# B&R Automation Studio project A2019059_Linka_Power_CP (part 11)

```iecst
(***************P4 - Funkčný test A************************************)

TYPE
	P4_FunkcnyTestA_typ : 	STRUCT
		IN : P4_FunkcnyTestA_IN_typ;
		OUT : P4_FunkcnyTestA_OUT_typ;
		PAR : P4_FunkcnyTestA_PAR_typ;
		STAV : P4_FunkcnyTestA_STAV_typ;
		Automat : BOOL;
		Manual : BOOL;
		Reset : BOOL;
		KoniecCyklu : BOOL;
		RR_TestovanieFunkcnehoTestu : BOOL;
		RR_ZapniOdpruzenieKontaktov : BOOL;
		RR_VysunKontaktyTestera : BOOL;
		RR_ZatvorTester : BOOL;
		RR_OtvorTester : BOOL;
	END_STRUCT;
	P4_FunkcnyTestA_IN_typ : 	STRUCT
		PritomnostPaletky_S10 : BOOL; (*RFID snímač na IO-linku*)
		PrecitaneCisloPaletky_S10 : USINT; (*RFID snímač na IO-linku*)
		HorneKontakty_VYSUNUTE_MS25 : BOOL;
		HorneKontakty_ZASUNUTE_MS23 : BOOL;
		SpodneKontakty_VYSUNUTE_MS33 : BOOL;
		SpodneKontakty_ZASUNUTE_MS31 : BOOL;
		Centrovanie_VYSUNUTE_MS29 : BOOL;
		Centrovanie_ZASUNUTE_MS27 : BOOL;
		TypSpodnychKontaktov_4F : BOOL;
		TypSpodnychKontaktov_5F_5H : BOOL;
	END_STRUCT;
	P4_FunkcnyTestA_OUT_typ : 	STRUCT
		ZasunStoper_YV163 : BOOL;
		HorneKontakty_VYSUN_YV178 : BOOL;
		HorneKontakty_ZASUN_YV177 : BOOL;
		OdpruzenieKontaktov_ZAPNI_YV179 : BOOL;
		OdpruzenieKontaktov_VYPNI_YV180 : BOOL;
		SpodneKontakty_VYSUN_YV182 : BOOL;
		SpodneKontakty_ZASUN_YV181 : BOOL;
		VysunCentrovanie_YV183 : BOOL;
		ZasunCentrovanie_YV184 : BOOL;
		KontaktyTestera_VYSUN_YV171 : BOOL;
		KOM_PLC_OdosliFotkyNaServer : BOOL;
		KOM_PLC_VymazFotky : BOOL;
	END_STRUCT;
	P4_FunkcnyTestA_PAR_typ : 	STRUCT
		SnimacPaletky_IOLinkInputs : ARRAY[1..10]OF USINT;
		IndexPaletky : USINT;
		IndexPaletky_STRING : STRING[2];
	END_STRUCT;
	P4_FunkcnyTestA_STAV_typ : 	STRUCT
		PoINIT : BOOL;
		KOM_PLC_OdoslanieFotiek_OK : BOOL;
		KOM_PLC_VymazanieFotiek_OK : BOOL;
		Vysledok_FV_Testu : STRING[2]; (*OK alebo NG*)
		PrebiehaVyvezeniePaletky : BOOL;
		Tester_ON : BOOL;
	END_STRUCT;
END_TYPE

(***************P4 - Funkčný test B************************************)

TYPE
	P4_FunkcnyTestB_typ : 	STRUCT
		IN : P4_FunkcnyTestB_IN_typ;
		OUT : P4_FunkcnyTestB_OUT_typ;
		PAR : P4_FunkcnyTestB_PAR_typ;
		STAV : P4_FunkcnyTestB_STAV_typ;
		Automat : BOOL;
		Manual : BOOL;
		Reset : BOOL;
		KoniecCyklu : BOOL;
		RR_TestovanieFunkcnehoTestu : BOOL;
		RR_ZapniOdpruzenieKontaktov : BOOL;
		RR_VysunKontaktyTestera : BOOL;
		RR_ZatvorTester : BOOL;
		RR_OtvorTester : BOOL;
	END_STRUCT;
	P4_FunkcnyTestB_IN_typ : 	STRUCT
		PritomnostPaletky_S11 : BOOL; (*RFID snímač na IO-linku*)
		PrecitaneCisloPaletky_S11 : USINT; (*RFID snímač na IO-linku*)
		HorneKontakty_VYSUNUTE_MS26 : BOOL;
		HorneKontakty_ZASUNUTE_MS24 : BOOL;
		SpodneKontakty_VYSUNUTE_MS34 : BOOL;
		SpodneKontakty_ZASUNUTE_MS32 : BOOL;
		Centrovanie_VYSUNUTE_MS30 : BOOL;
		Centrovanie_ZASUNUTE_MS28 : BOOL;
		TypSpodnychKontaktov_4F : BOOL;
		TypSpodnychKontaktov_5F_5H : BOOL;
	END_STRUCT;
	P4_FunkcnyTestB_OUT_typ : 	STRUCT
		ZasunStoper_YV164 : BOOL;
		HorneKontakty_VYSUN_YV186 : BOOL;
		HorneKontakty_ZASUN_YV185 : BOOL;
		OdpruzenieKontaktov_ZAPNI_YV187 : BOOL;
		OdpruzenieKontaktov_VYPNI_YV188 : BOOL;
		SpodneKontakty_VYSUN_YV190 : BOOL;
		SpodneKontakty_ZASUN_YV189 : BOOL;
		VysunCentrovanie_YV191 : BOOL;
		ZasunCentrovanie_YV192 : BOOL;
		KontaktyTestera_VYSUN_YV172 : BOOL;
		KOM_PLC_OdosliFotkyNaServer : BOOL;
		KOM_PLC_VymazFotky : BOOL;
		KOM_StanicaA_StartTestovania : BOOL;
	END_STRUCT;
	P4_FunkcnyTestB_PAR_typ : 	STRUCT
		SnimacPaletky_IOLinkInputs : ARRAY[1..10]OF USINT;
		IndexPaletky : USINT;
		IndexPaletky_STRING : STRING[2];
	END_STRUCT;
	P4_FunkcnyTestB_STAV_typ : 	STRUCT
		PoINIT : BOOL;
		KOM_PLC_OdoslanieFotiek_OK : BOOL;
		KOM_PLC_VymazanieFotiek_OK : BOOL;
		Vysledok_FV_Testu : STRING[2]; (*OK alebo NG*)
		PrebiehaVyvezeniePaletky : BOOL;
		Tester_ON : BOOL;
	END_STRUCT;
END_TYPE

(***************P4 - Etiketovacka*************************************)

TYPE
	P4_Etiketovacka_typ : 	STRUCT
		IN : P4_Etiketovacka_IN_typ;
		OUT : P4_Etiketovacka_OUT_typ;
		PAR : P4_Etiketovacka_PAR_typ;
		STAV : P4_Etiketovacka_STAV_typ;
		Automat : BOOL;
		Manual : BOOL;
		Reset : BOOL;
		KoniecCyklu : BOOL;
		ServoZdvihuEtiketovania_M28 : Axis_Servo;
		RR_TestovanieEtiketovania : BOOL;
		RR_VysunAplikator : BOOL;
		RR_ZapniPrisavanie : BOOL;
	END_STRUCT;
	P4_Etiketovacka_IN_typ : 	STRUCT
		PritomnostPaletky_S12 : BOOL; (*RFID snímač na IO-linku*)
		PrecitaneCisloPaletky_S12 : USINT; (*RFID snímač na IO-linku*)
		Centrovanie_VYSUNUTE_IS54 : BOOL;
		Centrovanie_ZASUNUTE_IS55 : BOOL;
		ZdvihEtiketovania_RefSnimac_IS59 : BOOL;
		Aplikator_VYSUNUTY_MS36 : BOOL;
		Aplikator_ZASUNUTY_MS35 : BOOL;
		SnimacVakuaPrisavaniaEtikety_S32 : BOOL;
		NapajanieTlaciarne_OK : BOOL;
		Tlaciaren_ERROR : BOOL;
		Tlaciaren_READY : BOOL;
		Tlaciaren_DochadzaPaska : BOOL;
		PritlakPaskyOdisteny_IS84 : BOOL;
	END_STRUCT;
	P4_Etiketovacka_OUT_typ : 	STRUCT
		ZasunStoper_YV165 : BOOL;
		VysunCentrovanie_YV166 : BOOL;
		ZasunCentrovanie_YV167 : BOOL;
		Aplikator_VYSUN_YV173 : BOOL;
		Prisavanie_ZAPNI_YV175 : BOOL;
		Prisavanie_VYPNI_YV176 : BOOL;
		OfukEtikety_ZAPNI_YV174 : BOOL;
		KOM_PLC_OdosliFotkyNaServer : BOOL;
		KOM_PLC_VymazFotky : BOOL;
		Tlaciaren_START_Tlace : BOOL;
		Tlaciaren_RESET_Poruchy : BOOL;
	END_STRUCT;
	P4_Etiketovacka_PAR_typ : 	STRUCT
		ServoZdvihu_ZadanaPozicia : LREAL;
		ServoZdvihu_JoggRychlost : REAL;
		SnimacPaletky_IOLinkInputs : ARRAY[1..10]OF USINT;
		IndexPaletky : USINT;
		IndexPaletky_STRING : STRING[2];
		IndexFotky : USINT;
	END_STRUCT;
	P4_Etiketovacka_STAV_typ : 	STRUCT
		PoINIT : BOOL;
		ServoZdvihu_PoziciaDosiahnuta : BOOL;
		ServoZvihu_LimitSnimace_BUSY : BOOL;
		ServoZdvihu_HomingOK : BOOL;
		ServoZdvihu_BUSY : BOOL;
		Zdvih_AktualnaPozicia : LREAL;
		Zdvih_AktualnyMoment : REAL;
		Zdvih_AktualnaRychlost : REAL;
		Zdvih_JoggLimitDosiahnuty : BOOL;
		KOM_PLC_OdoslanieFotiek_OK : BOOL;
		KOM_PLC_VymazanieFotiek_OK : BOOL;
		OdoslanieFotiek_OK : BOOL;
		OdoslanieFotiek_Error : BOOL;
		VymazanieFotiek_OK : BOOL;
		VymazanieFotiek_Error : BOOL;
		PrebiehaVyvezeniePaletky : BOOL;
		PowerCP_ZhodaQRkodu_OK : BOOL;
		Etiketa_ZhodaQRkodu_OK : BOOL;
		TestovaciaSekvencia_BUSY : BOOL;
	END_STRUCT;
END_TYPE

(******************SkrutkovacieSety***********************)

TYPE
	P1_SkrutkovaciSetM5_typ : 	STRUCT
		Automat : BOOL;
		Manual : BOOL;
		Reset : BOOL;
		UkoncenieCyklu : BOOL;
		SkrutkaM5_Pripravena : BOOL;
		SkrutkaM5_Odobrata : BOOL;
	END_STRUCT;
	P1_SkrutkovaciSetK30_typ : 	STRUCT
		Automat : BOOL;
		Manual : BOOL;
		Reset : BOOL;
		UkoncenieCyklu : BOOL;
		Cistenie : BOOL;
		CistenieUkoncene : BOOL;
		SkrutkaK30_Pripravena : BOOL;
		SkrutkaK30_Odobrata : BOOL;
	END_STRUCT;
	P1_SkrutkovaciSetM4_typ : 	STRUCT
		Automat : BOOL;
		Manual : BOOL;
		Reset : BOOL;
		UkoncenieCyklu : BOOL;
		Cistenie : BOOL;
		CistenieUkoncene : BOOL;
		SkrutkaM4_Pripravena : BOOL;
		SkrutkaM4_Odobrata : BOOL;
	END_STRUCT;
	P2_SkrutkovaciSetM6_typ : 	STRUCT
		Automat : BOOL;
		Manual : BOOL;
		Reset : BOOL;
		UkoncenieCyklu : BOOL;
		Cistenie : BOOL;
		CistenieUkoncene : BOOL;
		SkrutkaM6_Pripravena : BOOL;
		SkrutkaM6_Odobrata : BOOL;
	END_STRUCT;
	P2_SkrutkovaciSetM5_typ : 	STRUCT
		Automat : BOOL;
		Manual : BOOL;
		Reset : BOOL;
		UkoncenieCyklu : BOOL;
		Cistenie : BOOL;
		CistenieUkoncene : BOOL;
		SkrutkaM5_Pripravena : BOOL;
		SkrutkaM5_Odobrata : BOOL;
	END_STRUCT;
	P2_SkrutkovaciSetM4_typ : 	STRUCT
		Automat : BOOL;
		Manual : BOOL;
		Reset : BOOL;
		UkoncenieCyklu : BOOL;
		Cistenie : BOOL;
		CistenieUkoncene : BOOL;
		SkrutkaM4_Pripravena : BOOL;
		SkrutkaM4_Odobrata : BOOL;
	END_STRUCT;
	P2_SkrutkovaciSetMaticaM4_typ : 	STRUCT
		Automat : BOOL;
		Manual : BOOL;
		Reset : BOOL;
		UkoncenieCyklu : BOOL;
		MaticaM4_Pripravena : BOOL;
		MaticaM4_Odobrata : BOOL;
	END_STRUCT;
	P3_SkrutkovaciSetK40_typ : 	STRUCT
		Automat : BOOL;
		Manual : BOOL;
		Reset : BOOL;
		UkoncenieCyklu : BOOL;
		Cistenie : BOOL;
		CistenieUkoncene : BOOL;
		SkrutkaK40_Pripravena : BOOL;
		SkrutkaK40_Odobrata : BOOL;
	END_STRUCT;
	P3_SkrutkovaciSetM5_typ : 	STRUCT
		Automat : BOOL;
		Manual : BOOL;
		Reset : BOOL;
		UkoncenieCyklu : BOOL;
		Cistenie : BOOL;
		CistenieUkoncene : BOOL;
		SkrutkaM5_Pripravena : BOOL;
		SkrutkaM5_Odobrata : BOOL;
	END_STRUCT;
END_TYPE

(*******************Devlink*****************************)

TYPE
	StrukturaNovehoNazvuAdresara_typ : 	STRUCT
		LINKA : STRING[10]; (*Názov linky PowerCP*)
		PRACOVISKO : STRING[10]; (*ST1,ST2,ST3 .......*)
		ROK : STRING[10]; (*YYYY*)
		DATUM : STRING[10]; (*YYYY_MM_SS*)
	END_STRUCT;
	StrukturaNovehoNazvuSuboru_typ : 	STRUCT
		DATUM : STRING[10]; (*YYYY_MM_DD*)
		CAS : STRING[8]; (*HH_MM_SS*)
		SERIAL : STRING[30]; (*Kód modelu*)
		INDEX : STRING[2]; (*1,2,3 ......*)
		RESULT : STRING[5]; (*PASS alebo FAIL*)
		Pripona : STRING[5]; (*.jpg*)
	END_STRUCT;
END_TYPE

(**************Skrutkovacky***************************)

TYPE
	SkrutkovackaAtlasCopco_typ : 	STRUCT
		RESET_Poruchy : BOOL;
		RESET_Vysledkov : BOOL;
		START_Skrutkovania : BOOL;
		START_Utahovania : BOOL;
		Stav_VysledokPotvrdeny : BOOL;
		Stav_EmergencyStop : BOOL;
		Stav_READY_to_START : BOOL;
		Stav_MANUAL : BOOL;
		Stav_UtahovanieUkoncene : BOOL;
		Stav_VysledokUtahovania_OK : BOOL;
		Stav_VysledokUtahovania_NG : BOOL;
		Stav_SmerOtacania_VPRED : BOOL;
		Stav_BUSY : BOOL;
		Stav_ControlerSwitch_ON : BOOL;
		Stav_Station_READY : BOOL;
		Stav_NastrojPripojeny : BOOL;
		Stav_NastrojUtahuje : BOOL;
		Stav_CisloAktualnehoProgramu : USINT;
		CisloZadanehoProgramu : USINT;
		VyslednyReport : STRING[5];
	END_STRUCT;
END_TYPE

(**************Ateq Leakage Testery******************)

TYPE
	AteqTester_typ : 	STRUCT
		START_Testovania : BOOL;
		RESET_Vysledkov : BOOL;
		ZMEN_Program : BOOL;
		CitajParametreTestera : BOOL;
		Stav_RESET_DONE : BOOL;
		Stav_START_DONE : BOOL;
		Stav_ZmenaProgramu_DONE : BOOL;
		Stav_ERROR : BOOL;
		Stav_READY : BOOL;
		Stav_BUSY : BOOL;
		Stav_CitanieParametrov_OK : BOOL;
		Stav_CitanieParametrov_ERROR : BOOL;
		CisloZadanehoProgramu : UINT;
		CisloAktualnehoProgramu : UINT;
		VysledokTestovania_OK : BOOL;
		VysledokTestovania_NG : BOOL;
		Profinet_PLC_INPUTS : ARRAY[1..100]OF USINT;
		Profinet_PLC_OUTPUTS : ARRAY[1..100]OF USINT;
		ReadParameter_1 : UINT;
		ReadParameter_2 : UINT;
		ReadParameter_3 : UINT;
		ReadParameter_4 : UINT;
		ReadParameter_5 : DINT;
		PocetCitanychParametrov : USINT;
		IdentifikaciaParametra_1 : USINT;
		IdentifikaciaParametra_2 : USINT;
		IdentifikaciaParametra_3 : USINT;
		IdentifikaciaParametra_4 : USINT;
		CasPnenia : REAL;
		CasStabilizacie : REAL;
		TlakPlnenia : REAL;
		Tolerancia : REAL;
		TlakUniku : REAL;
	END_STRUCT;
END_TYPE

(***************Etiketa********************************)

TYPE
	Etiketa_typ : 	STRUCT
		LocationCode : STRING[2]; (*KK*)
		PartIdentNumber : STRING[7]; (*SSSSSSS*)
		ChangeIndex : STRING[2]; (*II*)
		ProductionYear : STRING[2]; (*JJ*)
		Manufactured : STRING[1]; (*H*)
		DayOfProduction : STRING[3]; (*TTT*)
		AssemblyLine : STRING[1]; (*M*)
		DayProductionCounter : STRING[5]; (*PPPPP*)
		SuplierNumber : STRING[6]; (*LLLLLL*)
		PlantCode : STRING[2]; (*NN*)
		DataMetrix : STRING[31]; (*Vytváram ho z kodu modelu na pracovisku etiketovania*)
		TypModelu : STRING[8];
		CountryCode : STRING[2];
		DatumVyroby : STRING[8]; (*02.03.20*)
	END_STRUCT;
END_TYPE

(***************Komunikácia zo serverom********************)

TYPE
	KOM_Server_typ : 	STRUCT
		CMD : KOM_Server_CMD_typ;
		INPUTS : KOM_Server_INPUTS_typ;
		OUTPUTS : KOM_Server_OUTPUTS_typ;
		STATUS : KOM_Server_STATUS_typ;
	END_STRUCT;
	KOM_Server_CMD_typ : 	STRUCT
		VyziadajStavPaletky_TYP1 : BOOL;
		PriradQRkodFiltra_TYP3 : BOOL;
		VyziadajCisloEtikety_TYP0 : BOOL;
		OdosliStavPaletky_TYP2 : BOOL;
	END_STRUCT;
	KOM_Server_INPUTS_typ : 	STRUCT
		TYP_Prikazu : STRING[1]; (*Typ*)
		CisloStanice : STRING[5]; (*Stanica*)
		CisloPaletky : STRING[10]; (*RFID paletky*)
		QRkodPowerCP : STRING[30]; (*Master number*)
		QRkodFiltra : STRING[30]; (*DPS1*)
		ID_Operatora : STRING[80]; (*Operator*)
		Report : STRING[4000]; (*DATA  - Oddelené bodkočiarkou*)
		StavPaletky : STRING[4]; (*PASS alebo FAIL*)
		IndexPaletky : USINT;
	END_STRUCT;
	KOM_Server_OUTPUTS_typ : 	STRUCT
		TYP_Prikazu : STRING[1]; (*Typ*)
		CisloStanice : STRING[5]; (*Stanica*)
		CisloPaletky : STRING[10]; (*RFID paletky*)
		QRkodPowerCP : STRING[30]; (*Master number*)
		QRkodFiltra : STRING[30]; (*DPS1*)
		ID_Operatora : STRING[8]; (*Operator*)
		CisloEtikety : STRING[31];
		DruhCinnostiNaPaletke : STRING[20]; (*PRD;ST1 alebo SMP;CAL;ST1 alebo RST;HVT;ST1*)
		PovolenieCinnostiNaPaletke : STRING[2]; (*OK alebo NG*)
	END_STRUCT;
	KOM_Server_STATUS_typ : 	STRUCT
		KomunikaciaUkoncena : BOOL;
		KomunikaciaError : BOOL;
	END_STRUCT;
END_TYPE

(***************Vysledné reporty***************************)

TYPE
	Reports_typ : 	STRUCT
		Kamery : ReportKamery_typ;
		Skrutkovacky : ReportSkrutkovacky_typ;
		Zvaranie : ReportZvarania_typ;
		LeakageTest : ReportLeakageTest_typ;
	END_STRUCT;
	ReportKamery_typ : 	STRUCT
		P1_CAM2_KontrolaPaletky : STRING[5]; (*Výtah*)
		P1_CAM4_KontrolaPinovDPS : STRING[5]; (*Výtah*)
		P1_CAM6_KontrolaPaletky : STRING[5]; (*Srobovanie*)
		P2_CAM1_KontrolaTesnenia : STRING[5];
		P2_CAM17_KontrolaPaletky : STRING[5]; (*Zakladanie tesnenia*)
		P2_CAM9_KontrolaPaletky : STRING[5]; (*Srobovanie matice*)
		P2_CAM10_KontrolaPaletky : STRING[5]; (*Srobovanie*)
		P2_CAM11_KontrolaZvaru : STRING[5]; (*Zvaranie*)
		P2_CAM11_KontrolaPowerCP : STRING[5]; (*Zvaranie*)
		P2_CAM12_KontrolaPaletky : STRING[5];
		P3_CAM13_KontrolaPaletky : STRING[5]; (*Srobovanie*)
		P4_CAM15_KontrolaPaletky : STRING[5]; (*Etiketovačka*)
		P4_CAM16_KontrolaPaletky : STRING[5]; (*Výtah*)
	END_STRUCT;
	ReportSkrutkovacky_typ : 	STRUCT
		Moment_ToleranciaMAX : ReportSrobov_MomentTolerMAX_typ;
		Moment_ToleranciaMIN : ReportSrobov_MomentTolerMIN_typ;
		Moment_NameranaHodnota : ReportSrobov_NameranyMoment_typ;
		Uhol_ToleranciaMAX : ReportSrobov_UholTolerMAX_typ;
		Uhol_ToleranciaMIN : ReportSrobov_UholTolerMIN_typ;
		Uhol_NameranaHodnota : ReportSrobov_NameranyUhol_typ;
		VyskaSkrutkovania : ReportSrobov_VyskaSkrutkov_typ;
		CasSkrutkovania : ReportSrobov_CasSkrutkov_typ;
		VyslednyReport : ReportSrobov_VyslednyReport_typ;
	END_STRUCT;
	ReportZvarania_typ : 	STRUCT
		Vyska : ReportZvarania_Vyska_typ;
		Moment : ReportZvarania_Moment_typ;
		Frekvencia : STRING[10];
		VyslednyReport : STRING[5];
	END_STRUCT;
	ReportZvarania_Vyska_typ : 	STRUCT
		LavyZvar : STRING[10];
		PravyZvar : STRING[10];
	END_STRUCT;
	ReportZvarania_Moment_typ : 	STRUCT
		LavyZvar : STRING[4];
		PravyZvar : STRING[4];
	END_STRUCT;
	ReportSrobov_MomentTolerMAX_typ : 	STRUCT
		P1_LavaSkrutkaK30 : STRING[10];
		P1_PravaSkrutkaK30 : STRING[10];
		P1_ZadnaSkrutkaM4 : STRING[10];
		P1_PrednaSkrutkaM4 : STRING[10];
		P1_SkrutkaDPS_M4 : STRING[10];
		P1_LavaSkrutkaM5 : STRING[10];
		P1_PravaSkrutkaM5 : STRING[10];
		P1_StrednaSkrutkaM5 : STRING[10];
		P2_MaticaM4 : STRING[10];
		P2_LavaSkrutkaM6 : STRING[10];
		P2_PravaSkrutkaM6 : STRING[10];
		P2_LavaSkrutkaM4 : STRING[10];
		P2_PravaSkrutkaM4 : STRING[10];
		P2_LavaSkrutkaM5 : STRING[10];
		P2_PravaSkrutkaM5 : STRING[10];
		P2_StrednaSkrutkaM4 : STRING[10];
		P3_SkrutkaK40 : STRING[10];
		P3_SkrutkaM5 : STRING[10];
	END_STRUCT;
	ReportSrobov_MomentTolerMIN_typ : 	STRUCT
		P1_LavaSkrutkaK30 : STRING[10];
		P1_PravaSkrutkaK30 : STRING[10];
		P1_ZadnaSkrutkaM4 : STRING[10];
		P1_PrednaSkrutkaM4 : STRING[10];
		P1_SkrutkaDPS_M4 : STRING[10];
		P1_LavaSkrutkaM5 : STRING[10];
		P1_PravaSkrutkaM5 : STRING[10];
		P1_StrednaSkrutkaM5 : STRING[10];
		P2_MaticaM4 : STRING[10];
		P2_LavaSkrutkaM6 : STRING[10];
		P2_PravaSkrutkaM6 : STRING[10];
		P2_LavaSkrutkaM4 : STRING[10];
		P2_PravaSkrutkaM4 : STRING[10];
		P2_LavaSkrutkaM5 : STRING[10];
		P2_PravaSkrutkaM5 : STRING[10];
		P2_StrednaSkrutkaM4 : STRING[10];
		P3_SkrutkaK40 : STRING[10];
		P3_SkrutkaM5 : STRING[10];
	END_STRUCT;
	ReportSrobov_NameranyMoment_typ : 	STRUCT
		P1_LavaSkrutkaK30 : STRING[10];
		P1_PravaSkrutkaK30 : STRING[10];
		P1_ZadnaSkrutkaM4 : STRING[10];
		P1_PrednaSkrutkaM4 : STRING[10];
		P1_SkrutkaDPS_M4 : STRING[10];
		P1_LavaSkrutkaM5 : STRING[10];
		P1_PravaSkrutkaM5 : STRING[10];
		P1_StrednaSkrutkaM5 : STRING[10];
		P2_MaticaM4 : STRING[10];
		P2_LavaSkrutkaM6 : STRING[10];
		P2_PravaSkrutkaM6 : STRING[10];
		P2_LavaSkrutkaM4 : STRING[10];
		P2_PravaSkrutkaM4 : STRING[10];
		P2_LavaSkrutkaM5 : STRING[10];
		P2_PravaSkrutkaM5 : STRING[10];
		P2_StrednaSkrutkaM4 : STRING[10];
		P3_SkrutkaK40 : STRING[10];
		P3_SkrutkaM5 : STRING[10];
	END_STRUCT;
	ReportSrobov_UholTolerMAX_typ : 	STRUCT
		P1_LavaSkrutkaK30 : STRING[10];
		P1_PravaSkrutkaK30 : STRING[10];
		P1_ZadnaSkrutkaM4 : STRING[10];
		P1_PrednaSkrutkaM4 : STRING[10];
		P1_SkrutkaDPS_M4 : STRING[10];
		P1_LavaSkrutkaM5 : STRING[10];
		P1_PravaSkrutkaM5 : STRING[10];
		P1_StrednaSkrutkaM5 : STRING[10];
		P2_MaticaM4 : STRING[10];
		P2_LavaSkrutkaM6 : STRING[10];
		P2_PravaSkrutkaM6 : STRING[10];
		P2_LavaSkrutkaM4 : STRING[10];
		P2_PravaSkrutkaM4 : STRING[10];
		P2_LavaSkrutkaM5 : STRING[10];
		P2_PravaSkrutkaM5 : STRING[10];
		P2_StrednaSkrutkaM4 : STRING[10];
		P3_SkrutkaK40 : STRING[10];
		P3_SkrutkaM5 : STRING[10];
	END_STRUCT;
	ReportSrobov_UholTolerMIN_typ : 	STRUCT
		P1_LavaSkrutkaK30 : STRING[10];
		P1_PravaSkrutkaK30 : STRING[10];
		P1_ZadnaSkrutkaM4 : STRING[10];
		P1_PrednaSkrutkaM4 : STRING[10];
		P1_SkrutkaDPS_M4 : STRING[10];
		P1_LavaSkrutkaM5 : STRING[10];
		P1_PravaSkrutkaM5 : STRING[10];
		P1_StrednaSkrutkaM5 : STRING[10];
		P2_MaticaM4 : STRING[10];
		P2_LavaSkrutkaM6 : STRING[10];
		P2_PravaSkrutkaM6 : STRING[10];
		P2_LavaSkrutkaM4 : STRING[10];
		P2_PravaSkrutkaM4 : STRING[10];
		P2_LavaSkrutkaM5 : STRING[10];
		P2_PravaSkrutkaM5 : STRING[10];
		P2_StrednaSkrutkaM4 : STRING[10];
		P3_SkrutkaK40 : STRING[10];
		P3_SkrutkaM5 : STRING[10];
	END_STRUCT;
	ReportSrobov_NameranyUhol_typ : 	STRUCT
		P1_LavaSkrutkaK30 : STRING[10];
		P1_PravaSkrutkaK30 : STRING[10];
		P1_ZadnaSkrutkaM4 : STRING[10];
		P1_PrednaSkrutkaM4 : STRING[10];
		P1_SkrutkaDPS_M4 : STRING[10];
		P1_LavaSkrutkaM5 : STRING[10];
		P1_PravaSkrutkaM5 : STRING[10];
		P1_StrednaSkrutkaM5 : STRING[10];
		P2_MaticaM4 : STRING[10];
		P2_LavaSkrutkaM6 : STRING[10];
		P2_PravaSkrutkaM6 : STRING[10];
		P2_LavaSkrutkaM4 : STRING[10];
		P2_PravaSkrutkaM4 : STRING[10];
		P2_LavaSkrutkaM5 : STRING[10];
		P2_PravaSkrutkaM5 : STRING[10];
		P2_StrednaSkrutkaM4 : STRING[10];
		P3_SkrutkaK40 : STRING[10];
		P3_SkrutkaM5 : STRING[10];
	END_STRUCT;
	ReportSrobov_VyskaSkrutkov_typ : 	STRUCT
		P1_LavaSkrutkaK30 : STRING[10];
		P1_PravaSkrutkaK30 : STRING[10];
		P1_ZadnaSkrutkaM4 : STRING[10];
		P1_PrednaSkrutkaM4 : STRING[10];
		P1_SkrutkaDPS_M4 : STRING[10];
		P1_LavaSkrutkaM5 : STRING[10];
		P1_PravaSkrutkaM5 : STRING[10];
		P1_StrednaSkrutkaM5 : STRING[10];
		P2_MaticaM4 : STRING[10];
		P2_LavaSkrutkaM6 : STRING[10];
		P2_PravaSkrutkaM6 : STRING[10];
		P2_LavaSkrutkaM4 : STRING[10];
		P2_PravaSkrutkaM4 : STRING[10];
		P2_LavaSkrutkaM5 : STRING[10];
		P2_PravaSkrutkaM5 : STRING[10];
		P2_StrednaSkrutkaM4 : STRING[10];
		P3_SkrutkaK40 : STRING[10];
		P3_SkrutkaM5 : STRING[10];
	END_STRUCT;
	ReportSrobov_CasSkrutkov_typ : 	STRUCT
		P1_LavaSkrutkaK30 : STRING[10];
		P1_PravaSkrutkaK30 : STRING[10];
		P1_ZadnaSkrutkaM4 : STRING[10];
		P1_PrednaSkrutkaM4 : STRING[10];
		P1_SkrutkaDPS_M4 : STRING[10];
		P1_LavaSkrutkaM5 : STRING[10];
		P1_PravaSkrutkaM5 : STRING[10];
		P1_StrednaSkrutkaM5 : STRING[10];
		P2_MaticaM4 : STRING[10];
		P2_LavaSkrutkaM6 : STRING[10];
		P2_PravaSkrutkaM6 : STRING[10];
		P2_LavaSkrutkaM4 : STRING[10];
		P2_PravaSkrutkaM4 : STRING[10];
		P2_LavaSkrutkaM5 : STRING[10];
		P2_PravaSkrutkaM5 : STRING[10];
		P2_StrednaSkrutkaM4 : STRING[10];
		P3_SkrutkaK40 : STRING[10];
		P3_SkrutkaM5 : STRING[10];
	END_STRUCT;
	ReportSrobov_VyslednyReport_typ : 	STRUCT
		P1_LavaSkrutkaK30 : STRING[5];
		P1_PravaSkrutkaK30 : STRING[5];
		P1_ZadnaSkrutkaM4 : STRING[5];
		P1_PrednaSkrutkaM4 : STRING[5];
		P1_SkrutkaDPS_M4 : STRING[5];
		P1_LavaSkrutkaM5 : STRING[5];
		P1_PravaSkrutkaM5 : STRING[5];
		P1_StrednaSkrutkaM5 : STRING[5];
		P2_MaticaM4 : STRING[5];
		P2_LavaSkrutkaM6 : STRING[5];
		P2_PravaSkrutkaM6 : STRING[5];
		P2_LavaSkrutkaM4 : STRING[5];
		P2_PravaSkrutkaM4 : STRING[5];
		P2_LavaSkrutkaM5 : STRING[5];
		P2_PravaSkrutkaM5 : STRING[5];
		P2_StrednaSkrutkaM4 : STRING[5];
		P3_SkrutkaK40 : STRING[5];
		P3_SkrutkaM5 : STRING[5];
	END_STRUCT;
	ReportLeakageTest_typ : 	STRUCT
		CasPlnenia : RepLeakTest_CasPlnenia_typ;
		CasStabilizacie : RepLeakTest_CasStabilizacie_typ;
		TlakPlnenia : RepLeakTest_TlakPlnenia_typ;
		TlakPritlaku : RepLeakTest_TlakPritlaku_typ;
		ToleranciaPritlaku_MIN : RepLeakTest_TolPritlakuMIN_typ;
		ToleranciaPritlaku_MAX : RepLeakTest_TolPritlakuMAX_typ;
		ToleranciaTlakUniku_MIN : RepLeakTest_TolTlakUnikuMIN_typ;
		ToleranciaTlakUniku_MAX : RepLeakTest_TolTlakUnikuMAX_typ;
		TlakUniku : RepLeakTest_TlakUniku_typ;
		Tolerancia : RepLeakTest_Tolerancia_typ;
		VyslednyReport : RepLeakTest_VyslednyReport_typ;
	END_STRUCT;
	RepLeakTest_CasPlnenia_typ : 	STRUCT
		StanicaA : STRING[10];
		StanicaB : STRING[10];
	END_STRUCT;
	RepLeakTest_CasStabilizacie_typ : 	STRUCT
		StanicaA : STRING[10];
		StanicaB : STRING[10];
	END_STRUCT;
	RepLeakTest_TlakPlnenia_typ : 	STRUCT
		StanicaA : STRING[10];
		StanicaB : STRING[10];
	END_STRUCT;
	RepLeakTest_TlakPritlaku_typ : 	STRUCT
		StanicaA : STRING[10];
		StanicaB : STRING[10];
	END_STRUCT;
	RepLeakTest_TolPritlakuMIN_typ : 	STRUCT
		StanicaA : STRING[10];
		StanicaB : STRING[10];
	END_STRUCT;
	RepLeakTest_TolPritlakuMAX_typ : 	STRUCT
		StanicaA : STRING[10];
		StanicaB : STRING[10];
	END_STRUCT;
	RepLeakTest_TlakUniku_typ : 	STRUCT
		StanicaA : STRING[10];
		StanicaB : STRING[10];
	END_STRUCT;
	RepLeakTest_TolTlakUnikuMIN_typ : 	STRUCT
		StanicaA : STRING[10];
		StanicaB : STRING[10];
	END_STRUCT;
	RepLeakTest_TolTlakUnikuMAX_typ : 	STRUCT
		StanicaA : STRING[10];
		StanicaB : STRING[10];
	END_STRUCT;
	RepLeakTest_Tolerancia_typ : 	STRUCT
		StanicaA : STRING[10];
		StanicaB : STRING[10];
	END_STRUCT;
	RepLeakTest_VyslednyReport_typ : 	STRUCT
		StanicaA : STRING[5];
		StanicaB : STRING[5];
	END_STRUCT;
END_TYPE

(***************Posielanie fotiek na server**********************)

TYPE
	FTP_Kamery_typ : 	STRUCT
		CMD : FTP_Kamery_CMD_typ;
		INPUTS : FTP_Kamery_INPUTS_typ;
		STATUS : FTP_Kamery_STATUS_typ;
	END_STRUCT;
	FTP_Kamery_CMD_typ : 	STRUCT
		OdosliFotku : BOOL;
		VymazFotku : BOOL;
	END_STRUCT;
	FTP_Kamery_INPUTS_typ : 	STRUCT
		QRkodPowerCP : STRING[30]; (*Master number*)
		Result : STRING[5]; (*PASS alebo FAIL*)
		IndexFotky : STRING[2];
	END_STRUCT;
	FTP_Kamery_STATUS_typ : 	STRUCT
		KomunikaciaUkoncena : BOOL;
		KomunikaciaError : BOOL;
		CisloPoruchy : USINT;
		AdresarPrazdny : BOOL;
	END_STRUCT;
END_TYPE

(***************Meranie taktime********************************)

TYPE
	Taktime_typ : 	STRUCT
		CMD : Taktime_CMD_typ;
		OUTPUTS : Taktime_OUTPUTS_typ;
	END_STRUCT;
	Taktime_CMD_typ : 	STRUCT
		START_Merania_1 : BOOL;
		ZAPIS_Hodnot_1 : BOOL;
		STOP_Merania_1 : BOOL;
		START_Merania_2 : BOOL;
		ZAPIS_Hodnot_2 : BOOL;
		STOP_Merania_2 : BOOL;
	END_STRUCT;
	Taktime_OUTPUTS_typ : 	STRUCT
		NameraneHodiny_1 : UINT;
		NameraneMinuty_1 : UINT;
		NameraneSekundy_1 : UINT;
		NameraneMilisekundy_1 : UINT;
		NameraneHodiny_2 : UINT;
		NameraneMinuty_2 : UINT;
		NameraneSekundy_2 : UINT;
		NameraneMilisekundy_2 : UINT;
	END_STRUCT;
END_TYPE
```

### KameryGlobal.typ
```iecst
(************Kamera 1*******************)

TYPE
	CAM1_typ : 	STRUCT
		CMD : CAM1_Commands_typ;
		PAR : CAM1_Parametre_typ;
		STAV : CAM1_Status_typ;
		RESULT : CAM1_Results_typ;
		Profinet_PLC_INPUTS : ARRAY[0..100]OF USINT;
		Profinet_PLC_OUTPUTS : ARRAY[0..3]OF USINT;
	END_STRUCT;
	CAM1_Commands_typ : 	STRUCT
		Triger : BOOL;
		OdosliFotku : BOOL;
		VymazFotku : BOOL;
	END_STRUCT;
	CAM1_Parametre_typ : 	STRUCT
		ResultFotky : STRING[5];
	END_STRUCT;
	CAM1_Status_typ : 	STRUCT
		BUSY : BOOL;
		SWITCH : BOOL;
		READY : BOOL;
		OLD_SWITCH : BOOL;
		Results_READY : BOOL;
		Command_READY : BOOL;
		Command_ERROR : BOOL;
		Command_AKCEPTOVANY : BOOL;
	END_STRUCT;
	CAM1_Results_typ : 	STRUCT
		PritomnTesnenia_OK : BOOL;
		ZalozenieTesnenia_OK : BOOL;
		PritomnPowerCP_5H5F : BOOL;
		PritomnPowerCP_4F : BOOL;
	END_STRUCT;
END_TYPE

(*********Kamera 2***********)

TYPE
	CAM2_typ : 	STRUCT
		CMD : CAM2_Commands_typ;
		PAR : CAM2_Parametre_typ;
		STAV : CAM2_Status_typ;
		RESULT : CAM2_Results_typ;
		Profinet_PLC_INPUTS : ARRAY[0..100]OF USINT;
		Profinet_PLC_OUTPUTS : ARRAY[0..3]OF USINT;
	END_STRUCT;
	CAM2_Commands_typ : 	STRUCT
		Triger : BOOL;
		OdosliFotku : BOOL;
		VymazFotku : BOOL;
	END_STRUCT;
	CAM2_Parametre_typ : 	STRUCT
		ResultFotky : STRING[5];
	END_STRUCT;
	CAM2_Status_typ : 	STRUCT
		READY : BOOL;
		BUSY : BOOL;
		SWITCH : BOOL;
		OLD_SWITCH : BOOL;
		Results_READY : BOOL;
		Command_READY : BOOL;
		Command_ERROR : BOOL;
		Command_AKCEPTOVANY : BOOL;
	END_STRUCT;
	CAM2_Results_typ : 	STRUCT
		Paletka : CAM2_Paletka_typ;
		PowerCP : CAM2_PowerCP_typ;
	END_STRUCT;
	CAM2_PowerCP_typ : 	STRUCT
		New_Member : USINT;
	END_STRUCT;
	CAM2_Paletka_typ : 	STRUCT
		Pritom_PowerCP_5F : BOOL;
		Pritom_PowerCP_4F : BOOL;
		Pritom_PowerCP_5H : BOOL;
		Pritom_Busbar_SpodnyLavy_5H : BOOL;
		Pritom_Busbar_SpodnyPravy_5H : BOOL;
		Pritom_KrytuBusbarov_5H : BOOL;
		Pritom_DPS_4F5F : BOOL;
		Pritom_Busbaru_Spodny_5F : BOOL;
		Pritom_Busbaru_Spodny_4F : BOOL;
		Pritom_Foamu_4F5F : BOOL;
		Pritomn_Skeletonu_4F5F : BOOL;
		Pritomn_Skeletonu_5H : BOOL;
		Nepritomn_TopCoveru_4F : BOOL;
		Nepritomn_TopCoveru_5F5H : BOOL;
		Pritomn_LavyMVcase : BOOL;
		Pritomn_PravyMVcase : BOOL;
		OsadeniePlastuDPS_OK : BOOL;
		KompletSpodneBusbary_OK : BOOL;
	END_STRUCT;
END_TYPE

(***********Kamera 3****************)

TYPE
	CAM3_typ : 	STRUCT
		CMD : CAM3_Commands_typ;
		PAR : CAM3_Parametre_typ;
		STAV : CAM3_Status_typ;
		RESULT : CAM3_Results_typ;
		Profinet_QRkod_Znaky : ARRAY[0..31]OF USINT;
		Profinet_PLC_INPUTS : ARRAY[0..100]OF USINT;
		Profinet_PLC_OUTPUTS : ARRAY[0..3]OF USINT;
	END_STRUCT;
	CAM3_Commands_typ : 	STRUCT
		Triger : BOOL;
		OdosliFotku : BOOL;
		VymazFotku : BOOL;
	END_STRUCT;
	CAM3_Parametre_typ : 	STRUCT
		ResultFotky : STRING[5];
	END_STRUCT;
	CAM3_Status_typ : 	STRUCT
		BUSY : BOOL;
		SWITCH : BOOL;
		READY : BOOL;
		OLD_SWITCH : BOOL;
		Results_READY : BOOL;
	END_STRUCT;
	CAM3_Results_typ : 	STRUCT
		Paletka : CAM3_Paletka_typ;
		PowerCP : CAM3_PowerCP_typ;
	END_STRUCT;
	CAM3_PowerCP_typ : 	STRUCT
		New_Member : USINT;
	END_STRUCT;
	CAM3_Paletka_typ : 	STRUCT
		CitanieQRkodu_DPS_OK : BOOL;
		PrecitanyQRkod_DPS : STRING[32];
	END_STRUCT;
END_TYPE

(***********Kamera 4******************)

TYPE
	CAM4_typ : 	STRUCT
		CMD : CAM4_Commands_typ;
		PAR : CAM4_Parametre_typ;
		STAV : CAM4_Status_typ;
		RESULT : CAM4_Results_typ;
		Profinet_PLC_INPUTS : ARRAY[0..100]OF USINT;
		Profinet_PLC_OUTPUTS : ARRAY[0..3]OF USINT;
	END_STRUCT;
	CAM4_Commands_typ : 	STRUCT
		Triger : BOOL;
		OdosliFotku : BOOL;
		VymazFotku : BOOL;
	END_STRUCT;
	CAM4_Parametre_typ : 	STRUCT
		ResultFotky : STRING[5];
	END_STRUCT;
	CAM4_Status_typ : 	STRUCT
		READY : BOOL;
		BUSY : BOOL;
		SWITCH : BOOL;
		OLD_SWITCH : BOOL;
		Results_READY : BOOL;
		Command_READY : BOOL;
		Command_ERROR : BOOL;
		Command_AKCEPTOVANY : BOOL;
	END_STRUCT;
	CAM4_Results_typ : 	STRUCT
		Paletka : CAM4_Paletka_typ;
		PowerCP : CAM4_PowerCP_typ;
	END_STRUCT;
	CAM4_PowerCP_typ : 	STRUCT
		New_Member : USINT;
	END_STRUCT;
	CAM4_Paletka_typ : 	STRUCT
		Pritomn_Pinu1_KrytDPS_4F5F : BOOL;
		Pritomn_Pinu2_KrytDPS_4F5F : BOOL;
		Pritomn_Pinu3_KrytDPS_4F5F : BOOL;
		Pritomn_Pinu4_KrytDPS_4F5F : BOOL;
		Pritomn_Pinu5_KrytDPS_4F5F : BOOL;
		Pritomn_Pinu6_KrytDPS_4F5F : BOOL;
		Pritom_DPS_4F5F : BOOL;
	END_STRUCT;
END_TYPE

(***********Kamera 5******************)

TYPE
	CAM5_typ : 	STRUCT
		CMD : CAM5_Commands_typ;
		PAR : CAM5_Parametre_typ;
		STAV : CAM5_Status_typ;
		RESULT : CAM5_Results_typ;
		Profinet_QRkod_Znaky : ARRAY[0..31]OF USINT;
		Profinet_PLC_INPUTS : ARRAY[0..100]OF USINT;
		Profinet_PLC_OUTPUTS : ARRAY[0..3]OF USINT;
	END_STRUCT;
	CAM5_Commands_typ : 	STRUCT
		Triger : BOOL;
		OdosliFotku : BOOL;
		VymazFotku : BOOL;
	END_STRUCT;
	CAM5_Parametre_typ : 	STRUCT
		ResultFotky : STRING[5];
	END_STRUCT;
	CAM5_Status_typ : 	STRUCT
		BUSY : BOOL;
		SWITCH : BOOL;
		READY : BOOL;
		OLD_SWITCH : BOOL;
		Results_READY : BOOL;
	END_STRUCT;
	CAM5_Results_typ : 	STRUCT
		Paletka : CAM5_Paletka_typ;
		PowerCP : CAM5_PowerCP_typ;
	END_STRUCT;
	CAM5_PowerCP_typ : 	STRUCT
		CitanieQRkodu_PowerCP_OK : BOOL;
		PrecitanyQRkod_PowerCP : STRING[32];
	END_STRUCT;
	CAM5_Paletka_typ : 	STRUCT
		New_Member : USINT;
	END_STRUCT;
END_TYPE

(***********Kamera 6********************)

TYPE
	CAM6_typ : 	STRUCT
		CMD : CAM6_Commands_typ;
		PAR : CAM6_Parametre_typ;
		STAV : CAM6_Status_typ;
		RESULT : CAM6_Results_typ;
		Profinet_PLC_INPUTS : ARRAY[0..100]OF USINT;
		Profinet_PLC_OUTPUTS : ARRAY[0..3]OF USINT;
	END_STRUCT;
	CAM6_Commands_typ : 	STRUCT
		Triger : BOOL;
		OdosliFotku : BOOL;
		VymazFotku : BOOL;
	END_STRUCT;
	CAM6_Parametre_typ : 	STRUCT
		ResultFotky : STRING[5];
	END_STRUCT;
	CAM6_Status_typ : 	STRUCT
		READY : BOOL;
		BUSY : BOOL;
		SWITCH : BOOL;
		OLD_SWITCH : BOOL;
		Results_READY : BOOL;
		Command_READY : BOOL;
		Command_ERROR : BOOL;
		Command_AKCEPTOVANY : BOOL;
	END_STRUCT;
	CAM6_Results_typ : 	STRUCT
		Paletka : CAM6_Paletka_typ;
		PowerCP : CAM6_PowerCP_typ;
	END_STRUCT;
	CAM6_PowerCP_typ : 	STRUCT
		Nepritom_LavyFoam_4F5F : BOOL;
		Nepritom_PravyFoam_4F5F : BOOL;
		Pritom_LavejSkrutkyK30 : BOOL;
		Pritom_PravejSkrutkyK30 : BOOL;
		Pritom_SkrutkyDPS_4F5F : BOOL;
		Nepritom_ZadnejSkrutkyM4_4F : BOOL;
		Nepritom_ZadnejSkrutkyM4_5F : BOOL;
		Nepritom_PrednejSkrutkyM4_4F : BOOL;
		Nepritom_PrednejSkrutkyM4_5F : BOOL;
		Pritom_LavejSkrutkyM5_5H : BOOL;
		Pritom_PravejSkrutkyM5_5H : BOOL;
		Pritom_StrednejSkrutkyM5_5H : BOOL;
	END_STRUCT;
	CAM6_Paletka_typ : 	STRUCT
		Pritom_SpodnychBusbarov_5H : BOOL;
		Pritom_KrytuBusbarov_5H : BOOL;
		Pritom_SpodnyBusbar_5F : BOOL;
		Pritom_SpodnyBusbar_4F : BOOL;
		Pritom_LavyFoam_4F5F : BOOL;
		Pritom_PravyFoam_4F5F : BOOL;
	END_STRUCT;
END_TYPE

(************Kamera 7*******************)

TYPE
	CAM7_typ : 	STRUCT
		CMD : CAM7_Commands_typ;
		PAR : CAM7_Parametre_typ;
		STAV : CAM7_Status_typ;
		RESULT : CAM7_Results_typ;
		Profinet_QRkod_Znaky : ARRAY[0..31]OF USINT;
		Profinet_PLC_INPUTS : ARRAY[0..100]OF USINT;
		Profinet_PLC_OUTPUTS : ARRAY[0..3]OF USINT;
	END_STRUCT;
	CAM7_Commands_typ : 	STRUCT
		Triger : BOOL;
		OdosliFotku : BOOL;
		VymazFotku : BOOL;
	END_STRUCT;
	CAM7_Parametre_typ : 	STRUCT
		ResultFotky : STRING[5];
	END_STRUCT;
	CAM7_Status_typ : 	STRUCT
		BUSY : BOOL;
		SWITCH : BOOL;
		READY : BOOL;
		OLD_SWITCH : BOOL;
		Results_READY : BOOL;
		Command_READY : BOOL;
		Command_ERROR : BOOL;
		Command_AKCEPTOVANY : BOOL;
	END_STRUCT;
	CAM7_Results_typ : 	STRUCT
		CitanieQRkodu_Filtra5H_OK : BOOL;
		PrecitanyQRkod_Filtra5H : STRING[32];
	END_STRUCT;
END_TYPE

(************Kamera 8********************)

TYPE
	CAM8_typ : 	STRUCT
		CMD : CAM8_Commands_typ;
		PAR : CAM8_Parametre_typ;
		STAV : CAM8_Status_typ;
		RESULT : CAM8_Results_typ;
		Profinet_QRkod_Znaky : ARRAY[0..31]OF USINT;
		Profinet_PLC_INPUTS : ARRAY[0..100]OF USINT;
		Profinet_PLC_OUTPUTS : ARRAY[0..3]OF USINT;
	END_STRUCT;
	CAM8_Commands_typ : 	STRUCT
		Triger : BOOL;
		OdosliFotku : BOOL;
		VymazFotku : BOOL;
	END_STRUCT;
	CAM8_Parametre_typ : 	STRUCT
		ResultFotky : STRING[5];
	END_STRUCT;
	CAM8_Status_typ : 	STRUCT
		BUSY : BOOL;
		SWITCH : BOOL;
		READY : BOOL;
		OLD_SWITCH : BOOL;
		Results_READY : BOOL;
	END_STRUCT;
	CAM8_Results_typ : 	STRUCT
		Paletka : CAM8_Paletka_typ;
		PowerCP : CAM8_PowerCP_typ;
	END_STRUCT;
	CAM8_PowerCP_typ : 	STRUCT
		CitanieQRkodu_PowerCP_OK : BOOL;
		PrecitanyQRkod_PowerCP : STRING[30];
	END_STRUCT;
	CAM8_Paletka_typ : 	STRUCT
		New_Member : USINT;
	END_STRUCT;
END_TYPE

(*************Kamera 9********************)

TYPE
	CAM9_typ : 	STRUCT
		CMD : CAM9_Commands_typ;
		PAR : CAM9_Parametre_typ;
		STAV : CAM9_Status_typ;
		RESULT : CAM9_Results_typ;
		Profinet_PLC_INPUTS : ARRAY[0..100]OF USINT;
		Profinet_PLC_OUTPUTS : ARRAY[0..3]OF USINT;
	END_STRUCT;
	CAM9_Commands_typ : 	STRUCT
		Triger : BOOL;
		OdosliFotku : BOOL;
		VymazFotku : BOOL;
	END_STRUCT;
	CAM9_Parametre_typ : 	STRUCT
		ResultFotky : STRING[5];
	END_STRUCT;
	CAM9_Status_typ : 	STRUCT
		BUSY : BOOL;
		SWITCH : BOOL;
		READY : BOOL;
		OLD_SWITCH : BOOL;
		Results_READY : BOOL;
	END_STRUCT;
	CAM9_Results_typ : 	STRUCT
		Paletka : CAM9_Paletka_typ;
		PowerCP : CAM9_PowerCP_typ;
	END_STRUCT;
	CAM9_PowerCP_typ : 	STRUCT
		NepritomMatice : BOOL;
		PritomnBusbaru_5H : BOOL;
	END_STRUCT;
	CAM9_Paletka_typ : 	STRUCT
		New_Member : USINT;
	END_STRUCT;
END_TYPE

(**************Kamera 10******************)

TYPE
	CAM10_typ : 	STRUCT
		CMD : CAM10_Commands_typ;
		PAR : CAM10_Parametre_typ;
		STAV : CAM10_Status_typ;
		RESULT : CAM10_Results_typ;
		Profinet_PLC_INPUTS : ARRAY[0..100]OF USINT;
		Profinet_PLC_OUTPUTS : ARRAY[0..3]OF USINT;
	END_STRUCT;
	CAM10_Commands_typ : 	STRUCT
		Triger : BOOL;
		OdosliFotku : BOOL;
		VymazFotku : BOOL;
	END_STRUCT;
	CAM10_Parametre_typ : 	STRUCT
		ResultFotky : STRING[5];
	END_STRUCT;
	CAM10_Status_typ : 	STRUCT
		BUSY : BOOL;
		SWITCH : BOOL;
		READY : BOOL;
		OLD_SWITCH : BOOL;
		Results_READY : BOOL;
		Command_READY : BOOL;
		Command_ERROR : BOOL;
		Command_AKCEPTOVANY : BOOL;
	END_STRUCT;
	CAM10_Results_typ : 	STRUCT
		Paletka : CAM10_Paletka_typ;
		PowerCP : CAM10_PowerCP_typ;
	END_STRUCT;
	CAM10_PowerCP_typ : 	STRUCT
		Pritomn_LavejSkrutkyM6_4F5F : BOOL;
		Pritomn_PravejSkrutkyM6_4F5F : BOOL;
		Pritomn_LavejM4_4F5F : BOOL;
		Pritomn_PravejM4_4F5F : BOOL;
		Pritomn_SkrutkyM4_Filtra_5H : BOOL;
		Pritomn_LavejSkrutkyM5_5H : BOOL;
		Pritomn_PravejSkrutkyM5_5H : BOOL;
	END_STRUCT;
	CAM10_Paletka_typ : 	STRUCT
		Pritomn_Busbarov_5F : BOOL;
		Pritomn_Busbarov_4F : BOOL;
		Pritomn_Busbarov_5H : BOOL;
		Pritomn_PowerCP_5H : BOOL;
		Pritomn_PowerCP_4F : BOOL;
		Pritomn_PowerCP_5F : BOOL;
	END_STRUCT;
END_TYPE

(**************Kamera 11*****************)

TYPE
	CAM11_typ : 	STRUCT
		CMD : CAM11_Commands_typ;
		PAR : CAM11_Parametre_typ;
		STAV : CAM11_Status_typ;
		RESULT : CAM11_Results_typ;
		Profinet_PLC_INPUTS : ARRAY[0..100]OF USINT;
		Profinet_PLC_OUTPUTS : ARRAY[0..3]OF USINT;
	END_STRUCT;
	CAM11_Commands_typ : 	STRUCT
		Triger : BOOL;
		OdosliFotku : BOOL;
		VymazFotku : BOOL;
	END_STRUCT;
	CAM11_Parametre_typ : 	STRUCT
		ResultFotky : STRING[5];
	END_STRUCT;
	CAM11_Status_typ : 	STRUCT
		BUSY : BOOL;
		SWITCH : BOOL;
		READY : BOOL;
		OLD_SWITCH : BOOL;
		Results_READY : BOOL;
		Command_READY : BOOL;
		Command_ERROR : BOOL;
		Command_AKCEPTOVANY : BOOL;
	END_STRUCT;
	CAM11_Results_typ : 	STRUCT
		Paletka : CAM11_Paletka_typ;
		PowerCP : CAM11_PowerCP_typ;
	END_STRUCT;
	CAM11_Paletka_typ : 	STRUCT
		New_Member : USINT;
	END_STRUCT;
	CAM11_PowerCP_typ : 	STRUCT
		Pritomn_PowerCP_4F : BOOL;
		Pritomn_PowerCP_5F : BOOL;
		Pritomn_PowerCP_5H : BOOL;
		Pritomn_LavyMVcase : BOOL;
		Pritomn_PravyMVcase : BOOL;
		LavyBusbar_Zvaranie_OK : BOOL;
		PravyBusbar_Zvaranie_OK : BOOL;
		Pritomn_TopCover_4F : BOOL;
		Pritomn_TopCover_5F : BOOL;
		Pritomn_TopCover_5H : BOOL;
	END_STRUCT;
END_TYPE

(***************Kamera 12*****************)

TYPE
	CAM12_typ : 	STRUCT
		CMD : CAM12_Commands_typ;
		PAR : CAM12_Parametre_typ;
		STAV : CAM12_Status_typ;
		RESULT : CAM12_Results_typ;
		Profinet_PLC_INPUTS : ARRAY[0..100]OF USINT;
		Profinet_PLC_OUTPUTS : ARRAY[0..3]OF USINT;
	END_STRUCT;
	CAM12_Commands_typ : 	STRUCT
		Triger : BOOL;
		OdosliFotku : BOOL;
		VymazFotku : BOOL;
	END_STRUCT;
	CAM12_Parametre_typ : 	STRUCT
		ResultFotky : STRING[5];
	END_STRUCT;
	CAM12_Status_typ : 	STRUCT
		BUSY : BOOL;
		SWITCH : BOOL;
		READY : BOOL;
		OLD_SWITCH : BOOL;
		Results_READY : BOOL;
		Command_READY : BOOL;
		Command_ERROR : BOOL;
		Command_AKCEPTOVANY : BOOL;
	END_STRUCT;
	CAM12_Results_typ : 	STRUCT
		Paletka : CAM12_Paletka_typ;
		PowerCP : CAM12_PowerCP_typ;
	END_STRUCT;
	CAM12_Paletka_typ : 	STRUCT
		Pritomn_TopCover_5H5F : BOOL;
		Pritomn_TopCover_4F : BOOL;
		Pritomn_LavyMVcase : BOOL;
		Pritomn_PravyMVcase : BOOL;
	END_STRUCT;
	CAM12_PowerCP_typ : 	STRUCT
		New_Member : USINT;
	END_STRUCT;
END_TYPE

(***************Kamera 13****************)

TYPE
	CAM13_typ : 	STRUCT
		CMD : CAM13_Commands_typ;
		PAR : CAM13_Parametre_typ;
		STAV : CAM13_Status_typ;
		RESULT : CAM13_Results_typ;
		Profinet_PLC_INPUTS : ARRAY[0..100]OF USINT;
		Profinet_PLC_OUTPUTS : ARRAY[0..3]OF USINT;
	END_STRUCT;
	CAM13_Commands_typ : 	STRUCT
		Triger : BOOL;
		OdosliFotku : BOOL;
		VymazFotku : BOOL;
	END_STRUCT;
	CAM13_Parametre_typ : 	STRUCT
		ResultFotky : STRING[5];
	END_STRUCT;
	CAM13_Status_typ : 	STRUCT
		BUSY : BOOL;
		SWITCH : BOOL;
		READY : BOOL;
		OLD_SWITCH : BOOL;
		Results_READY : BOOL;
		Command_READY : BOOL;
		Command_ERROR : BOOL;
		Command_AKCEPTOVANY : BOOL;
	END_STRUCT;
	CAM13_Results_typ : 	STRUCT
		Pritomn_SkrutkyK40_TopCover_4F5F : BOOL;
		Pritomn_SkrutkyM5_TopCover : BOOL;
	END_STRUCT;
END_TYPE

(***************Kamera 14*****************)

TYPE
	CAM14_typ : 	STRUCT
		CMD : CAM14_Commands_typ;
		PAR : CAM14_Parametre_typ;
		STAV : CAM14_Status_typ;
		RESULT : CAM14_Results_typ;
		Profinet_QRkod_Znaky : ARRAY[0..31]OF USINT;
		Profinet_PLC_INPUTS : ARRAY[0..100]OF USINT;
		Profinet_PLC_OUTPUTS : ARRAY[0..3]OF USINT;
	END_STRUCT;
	CAM14_Commands_typ : 	STRUCT
		Triger : BOOL;
		OdosliFotku : BOOL;
		VymazFotku : BOOL;
	END_STRUCT;
	CAM14_Parametre_typ : 	STRUCT
		ResultFotky : STRING[5];
	END_STRUCT;
	CAM14_Status_typ : 	STRUCT
		BUSY : BOOL;
		SWITCH : BOOL;
		READY : BOOL;
		OLD_SWITCH : BOOL;
		Results_READY : BOOL;
	END_STRUCT;
	CAM14_Results_typ : 	STRUCT
		Paletka : CAM14_Paletka_typ;
		PowerCP : CAM14_PowerCP_typ;
	END_STRUCT;
	CAM14_PowerCP_typ : 	STRUCT
		CitanieQRkodu_PowerCP_OK : BOOL;
		PrecitanyQRkod_PowerCP : STRING[32];
	END_STRUCT;
	CAM14_Paletka_typ : 	STRUCT
		New_Member : USINT;
	END_STRUCT;
END_TYPE

(****************Kamera 15***************)

TYPE
	CAM15_typ : 	STRUCT
		CMD : CAM15_Commands_typ;
		PAR : CAM15_Parametre_typ;
		STAV : CAM15_Status_typ;
		RESULT : CAM15_Results_typ;
		Profinet_QRkod_Znaky : ARRAY[0..31]OF USINT;
		Profinet_OCR_Znaky : ARRAY[0..31]OF USINT;
		Profinet_PLC_INPUTS : ARRAY[0..100]OF USINT;
		Profinet_PLC_OUTPUTS : ARRAY[0..3]OF USINT;
	END_STRUCT;
	CAM15_Commands_typ : 	STRUCT
		Triger : BOOL;
		OdosliFotku : BOOL;
		VymazFotku : BOOL;
	END_STRUCT;
	CAM15_Parametre_typ : 	STRUCT
		ResultFotky : STRING[5];
	END_STRUCT;
	CAM15_Status_typ : 	STRUCT
		BUSY : BOOL;
		SWITCH : BOOL;
		READY : BOOL;
		OLD_SWITCH : BOOL;
		Results_READY : BOOL;
		Command_READY : BOOL;
		Command_ERROR : BOOL;
		Command_AKCEPTOVANY : BOOL;
	END_STRUCT;
	CAM15_Results_typ : 	STRUCT
		Pritomn_Etikety : BOOL;
		Pritomn_LogoBMV : BOOL;
		Pritomn_Textu_PowerCP : BOOL;
		Pritomn_Textu_Panasonic : BOOL;
		Pritomn_Textu_SK : BOOL;
		CitanieQRkodu_Etikety_OK : BOOL;
		PrecitanyQRkod_Etikety : STRING[31];
		PrecitaneOCR_Etikety : STRING[32];
	END_STRUCT;
END_TYPE

(****************Kamera 16**************)

TYPE
	CAM16_typ : 	STRUCT
		CMD : CAM16_Commands_typ;
		PAR : CAM16_Parametre_typ;
		STAV : CAM16_Status_typ;
		RESULT : CAM16_Results_typ;
		Profinet_PLC_INPUTS : ARRAY[0..100]OF USINT;
		Profinet_PLC_OUTPUTS : ARRAY[0..3]OF USINT;
	END_STRUCT;
	CAM16_Commands_typ : 	STRUCT
		Triger : BOOL;
		OdosliFotku : BOOL;
		VymazFotku : BOOL;
	END_STRUCT;
	CAM16_Parametre_typ : 	STRUCT
		ResultFotky : STRING[5];
	END_STRUCT;
	CAM16_Status_typ : 	STRUCT
		BUSY : BOOL;
		SWITCH : BOOL;
		READY : BOOL;
		OLD_SWITCH : BOOL;
		Results_READY : BOOL;
		Command_READY : BOOL;
		Command_ERROR : BOOL;
		Command_AKCEPTOVANY : BOOL;
	END_STRUCT;
	CAM16_Results_typ : 	STRUCT
		New_Member : USINT;
		Paletka : CAM16_Paletka_typ;
		PowerCP : CAM16_PowerCP_typ;
	END_STRUCT;
	CAM16_Paletka_typ : 	STRUCT
		Pritomn_Busbarov_4F : BOOL;
		Pritomn_Busbarov_5F : BOOL;
		Pritomn_Busbarov_5H : BOOL;
		Pritomn_LavyMVcase : BOOL;
		Pritomn_PravyMVcase : BOOL;
		Pritomn_PowerCP : BOOL;
		PrazdnaPaletka : BOOL;
	END_STRUCT;
	CAM16_PowerCP_typ : 	STRUCT
		PritomnostSkrutky_K40 : BOOL;
		PritomnostSkrutky_M5 : BOOL;
	END_STRUCT;
END_TYPE

(*************Kamera 17*******************)

TYPE
	CAM17_typ : 	STRUCT
		CMD : CAM17_Commands_typ;
		PAR : CAM17_Parametre_typ;
		STAV : CAM17_Status_typ;
		RESULT : CAM17_Results_typ;
		Profinet_PLC_INPUTS : ARRAY[0..100]OF USINT;
		Profinet_PLC_OUTPUTS : ARRAY[0..3]OF USINT;
	END_STRUCT;
	CAM17_Commands_typ : 	STRUCT
		Triger : BOOL;
		OdosliFotku : BOOL;
		VymazFotku : BOOL;
	END_STRUCT;
	CAM17_Parametre_typ : 	STRUCT
		ResultFotky : STRING[5];
	END_STRUCT;
	CAM17_Status_typ : 	STRUCT
		BUSY : BOOL;
		SWITCH : BOOL;
		READY : BOOL;
		OLD_SWITCH : BOOL;
		Results_READY : BOOL;
		Command_READY : BOOL;
		Command_ERROR : BOOL;
		Command_AKCEPTOVANY : BOOL;
	END_STRUCT;
	CAM17_Results_typ : 	STRUCT
		Paletka : CAM17_Paletka_typ;
		PowerCP : CAM17_PowerCP_typ;
	END_STRUCT;
	CAM17_PowerCP_typ : 	STRUCT
		New_Member : USINT;
	END_STRUCT;
	CAM17_Paletka_typ : 	STRUCT
		Pritomn_TopCoveru_4F : BOOL;
		Pritomn_TopCoveru_5F : BOOL;
		Pritomn_TopCoveru_5H : BOOL;
		Pritomn_Busbary_5H : BOOL;
		Pritomn_Busbary_5F : BOOL;
		Pritomn_Busbary_4F : BOOL;
		Pritomn_LavyMVcase : BOOL;
		Pritomn_PravyMVcase : BOOL;
		Pritomn_PowerCP_4F : BOOL;
		Pritomn_PowerCP_5F : BOOL;
		Pritomn_PowerCP_5H : BOOL;
		PoziciaBusbarov4F5F_OK : BOOL;
		PoziciaBusbarov5H_OK : BOOL;
	END_STRUCT;
END_TYPE

(************Control Unit********************)

TYPE
	ControlUnit_typ : 	STRUCT
		Profinet_PLC_INPUTS : ARRAY[0..1]OF USINT;
		Stav_READY : BOOL;
	END_STRUCT;
END_TYPE
```

### Global.var - Global variables
```iecst
(**********Nastavenie času**************)
VAR
	DTSetTime_0 : DTSetTime;
	DTGetTime_0 : DTGetTime;
END_VAR
(**********Blikače*******************************)
VAR
	Blikac100ms : BOOL;
	Blikac200ms : BOOL;
	Blikac500ms : BOOL;
	Blikac1s : BOOL;
END_VAR
(**************Remanentné premenné*********)
VAR
	P1_RemPremenne : P1_RemPremenne_typ;
	P2_RemPremenne : P2_RemPremenne_typ;
	P34_RemPremenne : P34_RemPremenne_typ;
	MpRecipeXml_P1 : MpRecipeXml := (0);
	MpRecipeRegPar_P1 : MpRecipeRegPar := (0);
	MpRecipeUI_P1 : MpRecipeUI;
	P1_UlozPremenne : BOOL;
	P1_NacitajPremenne : BOOL;
	MpRecipeXml_P2 : MpRecipeXml := (0);
	MpRecipeRegPar_P2 : MpRecipeRegPar := (0);
	MpRecipeUI_P2 : MpRecipeUI;
	P2_UlozPremenne : BOOL;
	P2_NacitajPremenne : BOOL;
	MpRecipeXml_P34 : MpRecipeXml := (0);
	MpRecipeRegPar_P34 : MpRecipeRegPar := (0);
	MpRecipeUI_P34 : MpRecipeUI;
	P34_UlozPremenne : BOOL;
	P34_NacitajPremenne : BOOL;
END_VAR
VAR RETAIN
	P1_Skrutk_4F_LavaK30_Vysunutie : REAL;
	P1_Skrutk_4F_PravaK30_Vysunutie : REAL;
	P1_Skrutk_4F_ZadnaM4_Vysunutie : REAL;
	P1_Skrutk_4F_PrednaM4_Vysunutie : REAL;
	P1_Skrutk_4F_DPS_M4_Vysunutie : REAL;
	P1_Skrutk_5F_LavaK30_Vysunutie : REAL;
	P1_Skrutk_5F_PravaK30_Vysunutie : REAL;
	P1_Skrutk_5F_ZadnaM4_Vysunutie : REAL;
	P1_Skrutk_5F_PrednaM4_Vysunutie : REAL;
	P1_Skrutk_5F_DPS_M4_Vysunutie : REAL;
	P1_Skrutk_5H_LavaK30_Vysunutie : REAL;
	P1_Skrutk_5H_PravaK30_Vysunutie : REAL;
	P1_Skrutk_5H_LavaM5_Vysunutie : REAL;
	P1_Skrutk_5H_PravaM5_Vysunutie : REAL;
	P1_Skrutk_5H_StrednaM5_Vysunutie : REAL;
	P2_Skrutk_4F_LavaM6_Vysunutie : REAL;
	P2_Skrutk_4F_PravaM6_Vysunutie : REAL;
	P2_Skrutk_4F_LavaM4_Vysunutie : REAL;
	P2_Skrutk_4F_PravaM4_Vysunutie : REAL;
	P2_Skrutk_5F_LavaM6_Vysunutie : REAL;
	P2_Skrutk_5F_PravaM6_Vysunutie : REAL;
	P2_Skrutk_5F_LavaM4_Vysunutie : REAL;
	P2_Skrutk_5F_PravaM4_Vysunutie : REAL;
	P2_Skrutk_5H_LavaM5_Vysunutie : REAL;
	P2_Skrutk_5H_PravaM5_Vysunutie : REAL;
	P2_Skrutk_5H_StrednaM4_Vysunutie : REAL;
	P2_Maticovacka_5H_Vysunutie : REAL;
	P3_Skrutk_4F_StredK40_Vysunutie : REAL;
	P3_Skrutk_4F_StredM5_Vysunutie : REAL;
	P3_Skrutk_5F_StredK40_Vysunutie : REAL;
	P3_Skrutk_5F_StredM5_Vysunutie : REAL;
	P3_Skrutk_5H_StredM5_Vysunutie : REAL;
END_VAR
(*************Všeobecné premenné*************)
VAR
	FilterVizu_P1 : STRING[300];
	FilterVizu_P2 : STRING[300];
	FilterVizu_P34 : STRING[300];
	Vizu : Vizu_typ;
	P1_Vizu : P1_Vizu_typ;
	P2_Vizu : P2_Vizu_typ;
	P34_Vizu : P34_Vizu_typ;
END_VAR
VAR RETAIN
	Paletka : ARRAY[0..20] OF Paletka_typ;
END_VAR
VAR
	Etiketa : Etiketa_typ;
	Safety : Safety_typ;
	Linka : Linka_typ;
	Reports : Reports_typ;
	P1_Pracovisko : P1_Pracovisko_typ;
	SC_P1_Dopravniky : SequenceControlTyp;
	P1_Dopravniky : P1_Dopravniky_typ;
	SC_P1_SpodnyStoper : SequenceControlTyp;
	P1_SpodnyStoper : P1_SpodnyStoper_typ;
	SC_P1_Vytah : SequenceControlTyp;
	P1_Vytah : P1_Vytah_typ;
	SC_P1_StoperSrobovania : SequenceControlTyp;
	P1_StoperSrobovania : P1_StoperSrobovacky_typ;
	SC_P1_Srobovanie : SequenceControlTyp;
	P1_Srobovanie : P1_Srobovanie_typ;
	SC_P1_AkumulacnyStoper : SequenceControlTyp;
	P1_AkumulacnyStoper : P1_AkumulacnyStoper_typ;
	SC_P1_Robot : SequenceControlTyp;
	P1_Robot : P1_Robot_typ;
	P2_Pracovisko : P2_Pracovisko_typ;
	SC_P2_Dopravniky : SequenceControlTyp;
	P2_Dopravniky : P2_Dopravniky_typ;
	SC_P2_StoperZaklTesnenia : SequenceControlTyp;
	P2_StoperZaklTesnenia : P2_StoperZaklTesnenia_typ;
	SC_P2_ZakladacTesnenia : SequenceControlTyp;
	P2_ZakladacTesnenia : P2_ZakladacTesnenia_typ;
	SC_P2_StoperMaticovacky : SequenceControlTyp;
	P2_StoperMaticovacky : P2_StoperMaticovacky_typ;
	SC_P2_SkrutkovacMatic : SequenceControlTyp;
	P2_SkrutkovacMatic : P2_SkrutkovacMatic_typ;
	SC_P2_StoperSrobovania : SequenceControlTyp;
	P2_StoperSrobovania : P2_StoperSrobovania_typ;
	SC_P2_Srobovanie : SequenceControlTyp;
	P2_Srobovanie : P2_Srobovanie_typ;
	SC_P2_Robot : SequenceControlTyp;
	P2_Robot : P2_Robot_typ;
	SC_P2_StoperZvarania : SequenceControlTyp;
	P2_StoperZvarania : P2_StoperZvarania_typ;
	SC_P2_Zvaranie : SequenceControlTyp;
	P2_Zvaranie : P2_Zvaranie_typ;
	SC_P2_Cistenie : SequenceControlTyp;
	P2_Cistenie : P2_Cistenie_typ;
	P3_Pracovisko : P3_Pracovisko_typ;
	SC_P3_Dopravniky : SequenceControlTyp;
	P3_Dopravniky : P3_Dopravniky_typ;
	SC_P3_SpodnyStoper : SequenceControlTyp;
	P3_SpodnyStoper : P3_SpodnyStoper_typ;
	SC_P3_VstupnyStoper : SequenceControlTyp;
	P3_VstupnyStoper : P3_VstupnyStoper_typ;
	SC_P3_StoperSrobovania : SequenceControlTyp;
	P3_StoperSrobovania : P3_StoperSrobovania_typ;
	SC_P3_Srobovanie : SequenceControlTyp;
	P3_Srobovanie : P3_Srobovanie_typ;
	SC_P3_AkumulacnyStoper : SequenceControlTyp;
	P3_AkumulacnyStoper : P3_AkumulacnyStoper_typ;
	SC_P3_LeakageTestA : SequenceControlTyp;
	P3_LeakageTestA : P3_LeakageTestA_typ;
	AteqLeakageTester_A : AteqTester_typ;
	SC_P3_LeakageTestB : SequenceControlTyp;
	P3_LeakageTestB : P3_LeakageTestB_typ;
	AteqLeakageTester_B : AteqTester_typ;
	P4_Pracovisko : P4_Pracovisko_typ;
	SC_P4_Dopravniky : SequenceControlTyp;
	P4_Dopravniky : P4_Dopravniky_typ;
	SC_P4_Vytah : SequenceControlTyp;
	P4_Vytah : P4_Vytah_typ;
	SC_P4_FunkcnyTestA : SequenceControlTyp;
	P4_FunkcnyTestA : P4_FunkcnyTestA_typ;
	SC_P4_FunkcnyTestB : SequenceControlTyp;
	P4_FunkcnyTestB : P4_FunkcnyTestB_typ;
	SC_P4_Etiketovacka : SequenceControlTyp;
	P4_Etiketovacka : P4_Etiketovacka_typ;
END_VAR
(**********Príznaky**************************)
VAR
	P1_Srobovacky_VychodziaPozicia : BOOL;
	P2_Srobovacky_VychodziaPozicia : BOOL;
	P2_Srobov_ManipulaciaUkoncena : BOOL;
	P2_Zvaranie_ManipulaciaUkoncena : BOOL;
	P3_Srobovacky_VychodziaPozicia : BOOL;
	P3_LeakageTestA_VychodziaPozicia : BOOL;
	P3_LeakageTestB_VychodziaPozicia : BOOL;
	P4_FunkcnyTestA_VychodziaPozicia : BOOL;
	P4_FunkcnyTestB_VychodziaPozicia : BOOL;
	P4_Etiketovacka_VychodziaPozicia : BOOL;
	CasCakaniaNaDruhePracovisko : TIME;
	Cas_HVTester : TON;
	NameranyCas_InitTestera : TIME;
	NameranyCas_PoslanieQRkodu : TIME;
	NameranyCas_CelkovyCasTestovania : TIME;
	Cas_FunkcnyTestA : TON;
	Cas_FunkcnyTestB : TON;
	NameranyCasFunkcnehoTestuA : TIME;
	NameranyCasFunkcnehoTestuB : TIME;
	Cas_PresunuSkrutky : TON;
	NameranyCasPresunuSkrutky : TIME;
END_VAR
(*************Tracebility***********************)
VAR
	TRCB_P1_Vytah_ST1 : KOM_Server_typ;
	TRCB_P1_Srobovanie_ST2 : KOM_Server_typ;
	TRCB_P2_ZakladacTesnenia_ST3 : KOM_Server_typ;
	TRCB_P2_Maticovacka_ST4 : KOM_Server_typ;
	TRCB_P2_Srobovanie_ST5 : KOM_Server_typ;
	TRCB_P2_Zvaranie_ST6 : KOM_Server_typ;
	TRCB_P3_Srobovanie_ST7 : KOM_Server_typ;
	TRCB_P3_LeakageTestA_ST8A : KOM_Server_typ;
	TRCB_P3_LeakageTestB_ST8B : KOM_Server_typ;
	TRCB_P4_Etiketovacka_ST9 : KOM_Server_typ;
	TRCB_P4_Vytah_ST10 : KOM_Server_typ;
	TRCB_P1_Srobov_OpatovnyDopyt : BOOL;
	TRCB_P1_Srobov_PaletkaNG : BOOL;
	TRCB_P2_ZaklTesn_OpatovnyDopyt : BOOL;
	TRCB_P2_ZaklTesn_PaletkaNG : BOOL;
	TRCB_P2_Maticov_OpatovnyDopyt : BOOL;
	TRCB_P2_Maticov_PaletkaNG : BOOL;
	TRCB_P2_Srobov_OpatovnyDopyt : BOOL;
	TRCB_P2_Srobov_PaletkaNG : BOOL;
	TRCB_P2_Zvaranie_OpatovnyDopyt : BOOL;
	TRCB_P2_Zvaranie_PaletkaNG : BOOL;
	TRCB_P3_Srobov_OpatovnyDopyt : BOOL;
	TRCB_P3_Srobov_PaletkaNG : BOOL;
	TRCB_P3_LeakTestA_OpatovnyDopyt : BOOL;
	TRCB_P3_LeakTestA_PaletkaNG : BOOL;
	TRCB_P3_LeakTestB_OpatovnyDopyt : BOOL;
	TRCB_P3_LeakTestB_PaletkaNG : BOOL;
	TRCB_P4_Etiketov_OpatovnyDopyt : BOOL;
	TRCB_P4_Etiketov_PaletkaNG : BOOL;
	TRCB_P4_Vytah_OpatovnyDopyt : BOOL;
	TRCB_P4_Vytah_PaletkaNG : BOOL;
END_VAR
(***************Odosielanie fotiek na server**************************)
VAR
	FTP_CAM1 : FTP_Kamery_typ; (*ST3 - zakladanie tesnenia - kontrola tesnenia*)
	FTP_CAM2 : FTP_Kamery_typ; (*ST1 - výtah - kontrola paletky*)
	FTP_CAM3 : FTP_Kamery_typ; (*ST1 - výtah - kontrola QR kodu DPS modely 4F a 5F*)
	FTP_CAM4 : FTP_Kamery_typ; (*ST1 - výtah - kontrola krytu DPS modely 4F a 5F*)
	FTP_CAM5 : FTP_Kamery_typ; (*ST1 - výtah - kontrola QR kodu Power CP*)
	FTP_CAM6 : FTP_Kamery_typ; (*ST2 - srobovanie - kontrola paletky*)
	FTP_CAM7 : FTP_Kamery_typ; (*ST3 - zakladanie tesnenia - kontrola filtra 5H*)
	FTP_CAM8 : FTP_Kamery_typ; (*ST3 - zakladanie tesnenia - kontrola QR kodu Power CP*)
	FTP_CAM9 : FTP_Kamery_typ; (*ST4 - maticovacka - kontrola paletky*)
	FTP_CAM10 : FTP_Kamery_typ; (*ST5 - srobovanie - kontrola paletky*)
	FTP_CAM11 : FTP_Kamery_typ; (*ST6 - zváranie - kontrola Power CP*)
	FTP_CAM12 : FTP_Kamery_typ; (*ST6 - zváranie - kontrola paletky*)
	FTP_CAM13 : FTP_Kamery_typ; (*ST7 - srobovanie - kontrola paletky*)
	FTP_CAM14 : FTP_Kamery_typ; (*ST9 - etiketovacka - kontrola QR kodu Power CP*)
	FTP_CAM15 : FTP_Kamery_typ; (*ST9 - etiketovacka - kontrola etikety*)
	FTP_CAM16 : FTP_Kamery_typ; (*ST10 - vytah - kontrola paletky*)
	FTP_CAM17 : FTP_Kamery_typ; (*ST3 - zakladanie tesnenia - kontrola paletky*)
	FTP_DMP_CAM1 : FTP_Kamery_typ;
	FTP_DMP_CAM2 : FTP_Kamery_typ;
	FTP_DMP_CAM3 : FTP_Kamery_typ;
	FTP_DMP_CAM4 : FTP_Kamery_typ;
	FTP_DMP_CAM5 : FTP_Kamery_typ;
	FTP_DMP_CAM6 : FTP_Kamery_typ;
	FTP_DMP_CAM7 : FTP_Kamery_typ;
	FTP_DMP_CAM8 : FTP_Kamery_typ;
	FTP_DMP_CAM9 : FTP_Kamery_typ;
	FTP_DMP_CAM10 : FTP_Kamery_typ;
	FTP_DMP_CAM11 : FTP_Kamery_typ;
	FTP_DMP_CAM12 : FTP_Kamery_typ;
	FTP_DMP_CAM13 : FTP_Kamery_typ;
	FTP_DMP_CAM14 : FTP_Kamery_typ;
	FTP_DMP_CAM15 : FTP_Kamery_typ;
	FTP_DMP_CAM16 : FTP_Kamery_typ;
	FTP_DMP_CAM17 : FTP_Kamery_typ;
END_VAR
(***************MeranieTaktimePracovisk***********************)
VAR
	Taktime_Vytah_ST1 : Taktime_typ;
	Taktime_Srobovanie_ST2 : Taktime_typ;
	Taktime_ZakladacTesnenia_ST3 : Taktime_typ;
	Taktime_Maticovacka_ST4 : Taktime_typ;
	Taktime_Srobovanie_ST5 : Taktime_typ;
	Taktime_Zvaranie_ST6 : Taktime_typ;
	Taktime_Srobovanie_ST7 : Taktime_typ;
	Taktime_LeakageTestA_ST8A : Taktime_typ;
	Taktime_LeakageTestB_ST8B : Taktime_typ;
	Taktime_FunkcnyTestA : Taktime_typ;
	Taktime_FunkcnyTestB : Taktime_typ;
	Taktime_Etiketovacka_ST9 : Taktime_typ;
	Taktime_Vytah_ST10 : Taktime_typ;
END_VAR
(**************Vypnutie výsledkov kamier a skrutkovacov******************)
VAR
	P1_Vytah_KAM_Result_OFF : BOOL;
	P1_Vytah_KAM_Result_Ignoruj : BOOL;
	P1_Srobov_KAM_Result_OFF : BOOL;
	P1_Srobov_KAM_Result_OK : BOOL;
	P1_Srobov_KAM_Result_NG : BOOL;
	P1_Srobov_K30_Result_OFF : BOOL;
	P1_Srobov_CakaNaKameru : BOOL;
	P1_Srobov_M5_Result_OFF : BOOL;
	P1_Srobov_M4_Result_OFF : BOOL;
	P2_ZaklTesn_KAM_Result_OFF : BOOL;
	P2_ZaklTesn_KAM_Result_Ignoruj : BOOL;
	P2_Maticov_KAM_Result_OFF : BOOL;
	P2_Maticov_KAM_Result_Ignoruj : BOOL;
	P2_Maticov_MaticaM4_Result_OFF : BOOL;
	P2_Maticov_CakaNaKameru : BOOL;
	P2_Maticov_KAM_Result_OK : BOOL;
	P2_Maticov_KAM_Result_NG : BOOL;
	P2_Srobov_KAM_Result_OFF : BOOL;
	P2_Srobov_KAM_Result_Ignoruj : BOOL;
	P2_Srobov_CakaNaKameru : BOOL;
	P2_Srobov_M4_Result_OFF : BOOL;
	P2_Srobov_M5_Result_OFF : BOOL;
	P2_Srobov_M6_Result_OFF : BOOL;
	P2_Srobov_KAM_Result_OK : BOOL;
	P2_Srobov_KAM_Result_NG : BOOL;
	P2_Zvaranie_KAM_Result_OFF : BOOL;
	P2_Zvaranie_KAM_Result_NG : BOOL;
	P2_Zvaranie_KAM_Result_OK : BOOL;
	P2_Zvaranie_CakaNaKameru : BOOL;
	P3_Srobov_KAM_Result_OFF : BOOL;
	P3_Srobov_KAM_Result_Ignoruj : BOOL;
	P3_Srobov_CakaNaKameru : BOOL;
	P3_Srobov_K40_Result_OFF : BOOL;
	P3_Srobov_M5_Result_OFF : BOOL;
	P3_HVTest_OTVOR : BOOL;
	P3_HVTest_ZATVOR : BOOL;
	P4_Etiketov_KAM_Result_OFF : BOOL;
	P4_Etiketov_KAM_Result_Ignoruj : BOOL;
	P4_Etiketov_KAM_Result_OK : BOOL;
	P4_Etiketov_KAM_Result_NG : BOOL;
	P4_Etiketov_CakaNaKameru : BOOL;
	P4_Vytah_KAM_Result_OFF : BOOL;
	P4_Vytah_CakaNaKameru : BOOL;
	P4_Vytah_KAM_Result_NG : BOOL;
	P4_Vytah_KAM_Result_Ignoruj : BOOL;
	P4_Vytah_KAM_Result_OK : BOOL;
	P4_FunkcnyTestA_ZATVOR : BOOL;
	P4_FunkcnyTestA_OTVOR : BOOL;
	P4_FunkcnyTestB_ZATVOR : BOOL;
	P4_FunkcnyTestB_OTVOR : BOOL;
	Kamery_PAUZA : BOOL;
END_VAR
```

### KameryGlobal.var
```iecst
(*****Pracovisko 1*********)
VAR
	CAM2 : CAM2_typ; (*P1_ST1_Vytah - kontrola kusov na paletke*)
	CAM3 : CAM3_typ; (*P1_ST1_Vytah - kontrola QR kódu DPS*)
	CAM4 : CAM4_typ; (*P1_ST1_Vytah - kontrola klipov krytu DPS*)
	CAM5 : CAM5_typ; (*P1_ST1_Vytah - kontrola QR kódu PowerCP*)
	CAM6 : CAM6_typ; (*P1_ST2_StoperSkrutkovania - Kontrola paletky*)
END_VAR
(******Pracovisko 2**********)
VAR
	CAM1 : CAM1_typ; (*P2_ST1_ZaklTesnenia - Kontrola tesnenia a QR kódu Power CP*)
	CAM7 : CAM7_typ; (*P2_ST1_StoperZaklTesnenia - Kontrola Power CP a QR kódu filtra*)
	CAM8 : CAM8_typ; (*P2_ST1_StoperZaklTesnenia - Kontrola spodného QR kódu Power CP*)
	CAM9 : CAM9_typ; (*P2_ST2_StoperMaticovacky - Kontrola paletky*)
	CAM10 : CAM10_typ; (*P2_ST3_StoperSkrutkovania - Kontrola paletky*)
	CAM11 : CAM11_typ; (*P2_ST4_StoperZvarania - Kontrola pravého MV case*)
	CAM12 : CAM12_typ; (*P2_ST4_StoperZvarania - Kontrola lavého MV case a Power CP*)
	CAM17 : CAM17_typ; (*P2_ST1_StoperZaklTesnenia - Kontrola paletky*)
END_VAR
(*******Pracovisko 3**************)
VAR
	CAM13 : CAM13_typ; (*P3_ST1_*)
END_VAR
(********Pracovisko 4*************)
VAR
	CAM14 : CAM14_typ; (*P4_ST3_*)
	CAM15 : CAM15_typ; (*P4_ST3_*)
	CAM16 : CAM16_typ; (*P4_ST4_*)
END_VAR
(*********Control Unit********************)
VAR
	ControlUnit : ControlUnit_typ;
END_VAR
```

### Package Logical/Libraries - Global libraries

### Library Logical/Libraries/SC (IEC)

#### Types.typ - Exported data types
```iecst
TYPE
	SequenceControlTyp : 	STRUCT
		StepName : STRING[80];
		Step : UINT;
		Switch1 : BOOL;
		Switch2 : BOOL;
		Switch3 : BOOL;
		ResetStep : BOOL;
		LastStep : BOOL;
		IdleTime : TON;
		AlarmTime : TON;
	END_STRUCT;
END_TYPE
```

#### SC.fun - Exported functions and function blocks
```iecst
FUNCTION SequenceControl : BOOL
	VAR_IN_OUT
		SC : SequenceControlTyp;
	END_VAR
END_FUNCTION
```

#### SequenceControl.st
```iecst
(* TODO: Add your comment here *)
FUNCTION SequenceControl

	IF SC.ResetStep THEN
		brsmemset(ADR(SC.StepName),0,SIZEOF(SC.StepName));
		SC.Switch1:= FALSE;
		SC.Switch2:= FALSE;
		SC.Switch3:= FALSE;
		SC.IdleTime.IN:= FALSE;
		SC.AlarmTime.IN:= FALSE;
		SC.ResetStep:= FALSE;
	END_IF

	IF SC.LastStep THEN
		brsmemset(ADR(SC.StepName),0,SIZEOF(SC.StepName));
		SC.Switch1:= FALSE;
		SC.Switch2:= FALSE;
		SC.Switch3:= FALSE;
		SC.IdleTime.IN:= FALSE;
		SC.AlarmTime.IN:= FALSE;
		SC.Step:= 0;
		SC.LastStep:= FALSE;
	END_IF

	//Volanie časovačov//
	SC.AlarmTime();
	SC.IdleTime();

END_FUNCTION
```

### Library Logical/Libraries/AxisLib (IEC)

#### Types.typ - Exported data types
```iecst
TYPE
	ServoCommand_typ : 	STRUCT
		ENABLE : BOOL;
		POWER : BOOL;
		HOME : BOOL;
		JoggVPRED : BOOL;
		JoggVZAD : BOOL;
		JoggLimit_ACTIVE : BOOL;
		MoveAbsolute : BOOL;
		MoveVelocity : BOOL;
		MoveAdditive : BOOL;
		MoveTorque : BOOL;
		STOP : BOOL;
		ErrorRESET : BOOL;
		UvolniBRZDU : BOOL;
		ZabrzdiBRZDU : BOOL;
		UpdatePAR : BOOL;
	END_STRUCT;
	ServoParametre_typ : 	STRUCT
		Acceleration : REAL;
		Deceleration : REAL;
		Velocity : REAL;
		Position : LREAL;
		AdditivePosition : LREAL;
		MoveDirection : USINT; (*0 - chod vpred, 1 - chod vzad, 10 - chod obojsmerný*)
		JoggAcceleration : REAL;
		JoggDeceleration : REAL;
		JoggVelocity : REAL;
		JoggPoziciaLimitVPRED : LREAL;
		JoggPoziciaLimitVZAD : LREAL;
		Torque : REAL;
		TorqueVelocity : REAL;
		TorqueAcceleration : REAL;
		TorqueRamp : REAL;
		StopDeceleration : REAL; (*Rampa zastavenia po Stop*)
		ZmenaRychlosti : REAL; (*Rozsah od 0.0 do 2.0 po 0.0001, 1.0 - 100%, 2.0 - 200% *)
		ZmenaRampy : REAL; (*Rozsah od 0.1 do 2.0 po 0.0001, 1.0 - 100%, 2.0 - 200%*)
	END_STRUCT;
	ServoStatus_typ : 	STRUCT
		ReadyToPower_ON : BOOL;
		Communication_READY : BOOL;
		Power_ON : BOOL;
		ActualPosition : LREAL;
		ActualVelocity : REAL;
		ActualTorque : REAL;
		MoveAbsolute_DONE : BOOL;
		MoveAdditive_DONE : BOOL;
		Rychlost_Dosiahnuta : BOOL;
		JoggLimit_Dosiahnuty : BOOL;
		Torque_Dosiahnuty : BOOL;
		Homing_OK : BOOL;
		Homing_BUSY : BOOL;
		MoveAbsolute_BUSY : BOOL;
		MoveVelocity_BUSY : BOOL;
		MoveAdditive_BUSY : BOOL;
		MoveTorque_BUSY : BOOL;
		Jogging_BUSY : BOOL;
		UpdatePAR_DONE : BOOL;
		STOP_ACTIVE : BOOL;
		EnableSwitch_ACTIVE : BOOL;
		HomingSwitch_ACTIVE : BOOL;
		PositiveLimitSwitch_ACTIVE : BOOL;
		NegativeLimitSwitch_ACTIVE : BOOL;
		Torque_AxisLimit_ACTIVE : BOOL;
		ERROR : BOOL;
		ERROR_ID : DINT;
		UvolnenieBrzdy_DONE : BOOL;
		ZabrzdenieBrzdy_DONE : BOOL;
	END_STRUCT;
	ServoErrorDetail_typ : 	STRUCT
		Power_Error : BOOL;
		Power_ErrorID : DINT;
		Home_Error : BOOL;
		Home_ErrorID : DINT;
		JoggLimit_Error : BOOL;
		JoggLimit_ErrorID : DINT;
		Jogg_Error : BOOL;
		Jogg_ErrorID : DINT;
		MoveAbsolute_Error : BOOL;
		MoveAbsolute_ErrorID : DINT;
		MoveAdditive_Error : BOOL;
		MoveAdditive_ErrorID : DINT;
		MoveVelocity_Error : BOOL;
		MoveVelocity_ErrorID : DINT;
		MoveTorque_Error : BOOL;
		MoveTorque_ErrorID : DINT;
		Stop_Error : BOOL;
		Stop_ErrorID : DINT;
		BreakOperation_Error : BOOL;
		BreakOperation_ErrorID : DINT;
	END_STRUCT;
	ServoHomeParametre_typ : 	STRUCT
		Position : LREAL; (*Offset od home pozície, alebo offset od absolutneho snímača*)
		StartVelocity : REAL; (*Rýchlosť hladanie snímača*)
		HomingVelocity : REAL; (*Rýchlosť zostupu zo snímača*)
		Acceleration : REAL;
		HomeTorque : REAL; (*Moment na ktorom servo zastane a znuluje sa*)
		HomingOffset : LREAL; (*Offset od homing pozície*)
		HomingMode : USINT; (*0 - direct, 1 - referenčný snímač, 2 - limitný snímač, 3 - absolutný snímač, 4 - moment*)
	END_STRUCT;
	ServoInternal_typ : 	STRUCT
		MC_Power_0 : MC_Power;
		MC_ReadAxisInfo_0 : MC_ReadAxisInfo;
		MC_Home_0 : MC_Home;
		MC_ReadAxisError_0 : MC_ReadAxisError;
		MC_ReadStatus_0 : MC_ReadStatus;
		MC_BR_JogLimitPosition_0 : MC_BR_JogLimitPosition;
		MC_MoveAbsolute_0 : MC_MoveAbsolute;
		MC_MoveAdditive_0 : MC_MoveAdditive;
		MC_MoveVelocity_0 : MC_MoveVelocity;
		MC_Reset_0 : MC_Reset;
		MC_TorqueControl_0 : MC_TorqueControl; (*Iba pre servo*)
		MC_Stop_0 : MC_Stop;
		MC_BR_BrakeOperation_0 : MC_BR_BrakeOperation;
		MC_ReadActualPosition_0 : MC_ReadActualPosition;
		MC_ReadActualVelocity_0 : MC_ReadActualVelocity;
		MC_ReadActualTorque_0 : MC_ReadActualTorque; (*Iba pre servo*)
		MC_SetOverride_0 : MC_SetOverride;
		MC_BR_JogVelocity_0 : MC_BR_JogVelocity;
		MC_BR_InitHome_AcpAx_0 : MC_BR_InitHome_AcpAx;
		Home_STEP : USINT;
		CasTorque : TON;
	END_STRUCT;
	KrokacCommand_typ : 	STRUCT
		ENABLE : BOOL;
		POWER : BOOL;
		HOME : BOOL;
		JoggVPRED : BOOL;
		JoggVZAD : BOOL;
		JoggLimit_ACTIVE : BOOL;
		MoveAbsolute : BOOL;
		MoveVelocity : BOOL;
		MoveAdditive : BOOL;
		STOP : BOOL;
		ErrorRESET : BOOL;
		UvolniBRZDU : BOOL;
		ZabrzdiBRZDU : BOOL;
		UpdatePAR : BOOL;
	END_STRUCT;
	KrokacParametre_typ : 	STRUCT
		Acceleration : REAL;
		Deceleration : REAL;
		Velocity : REAL;
		Position : LREAL;
		AdditivePosition : LREAL;
		MoveDirection : USINT; (*0 - chod vpred, 1 - chod vzad, 10 - chod obojsmerný*)
		JoggAcceleration : REAL;
		JoggDeceleration : REAL;
		JoggVelocity : REAL;
		JoggPoziciaLimitVPRED : LREAL;
		JoggPoziciaLimitVZAD : LREAL;
		StopDeceleration : REAL; (*Rampa zastavenia po Stop*)
		ZmenaRychlosti : REAL; (*Rozsah od 0.0 do 2.0 po 0.0001, 1.0 - 100%, 2.0 - 200% *)
		ZmenaRampy : REAL; (*Rozsah od 0.1 do 2.0 po 0.0001, 1.0 - 100%, 2.0 - 200%*)
	END_STRUCT;
	KrokacStatus_typ : 	STRUCT
		ReadyToPower_ON : BOOL;
		Communication_READY : BOOL;
		Power_ON : BOOL;
		ActualPosition : LREAL;
		ActualVelocity : REAL;
		MoveAbsolute_DONE : BOOL;
		MoveAdditive_DONE : BOOL;
		Rychlost_Dosiahnuta : BOOL;
		JoggLimit_Dosiahnuty : BOOL;
		Homing_OK : BOOL;
		Homing_BUSY : BOOL;
		MoveAbsolute_BUSY : BOOL;
		MoveVelocity_BUSY : BOOL;
		MoveAdditive_BUSY : BOOL;
		Jogging_BUSY : BOOL;
		UpdatePAR_DONE : BOOL;
		STOP_ACTIVE : BOOL;
		EnableSwitch_ACTIVE : BOOL;
		HomingSwitch_ACTIVE : BOOL;
		PositiveLimitSwitch_ACTIVE : BOOL;
		NegativeLimitSwitch_ACTIVE : BOOL;
		ERROR : BOOL;
		ERROR_ID : DINT;
		UvolnenieBrzdy_DONE : BOOL;
		ZabrzdenieBrzdy_DONE : BOOL;
	END_STRUCT;
	KrokacErrorDetail_typ : 	STRUCT
		Power_Error : BOOL;
		Power_ErrorID : DINT;
		Home_Error : BOOL;
		Home_ErrorID : DINT;
		JoggLimit_Error : BOOL;
		JoggLimit_ErrorID : DINT;
		Jogg_Error : BOOL;
		Jogg_ErrorID : DINT;
		MoveAbsolute_Error : BOOL;
		MoveAbsolute_ErrorID : DINT;
		MoveAdditive_Error : BOOL;
		MoveAdditive_ErrorID : DINT;
		MoveVelocity_Error : BOOL;
		MoveVelocity_ErrorID : DINT;
		Stop_Error : BOOL;
		Stop_ErrorID : DINT;
		BreakOperation_Error : BOOL;
		BreakOperation_ErrorID : DINT;
		HomeSetup_Error : BOOL;
		HomeSetup_ErrorID : DINT;
	END_STRUCT;
	KrokacHomeParametre_typ : 	STRUCT
		Position : LREAL; (*Offset od home pozície*)
		StartVelocity : REAL; (*Rýchlosť hladanie snímača*)
		HomingVelocity : REAL; (*Rýchlosť zostupu zo snímača*)
		Acceleration : REAL;
		HomingMode : USINT; (*0 - direct, 1 - referenčný snímač, 2 - limitný snímač*)
	END_STRUCT;
	KrokacInternal_typ : 	STRUCT
		MC_Power_0 : MC_Power;
		MC_ReadAxisInfo_0 : MC_ReadAxisInfo;
		MC_Home_0 : MC_Home;
		MC_ReadAxisError_0 : MC_ReadAxisError;
		MC_ReadStatus_0 : MC_ReadStatus;
		MC_BR_JogLimitPosition_0 : MC_BR_JogLimitPosition;
		MC_MoveAbsolute_0 : MC_MoveAbsolute;
		MC_MoveAdditive_0 : MC_MoveAdditive;
		MC_MoveVelocity_0 : MC_MoveVelocity;
		MC_Reset_0 : MC_Reset;
		MC_Stop_0 : MC_Stop;
		MC_BR_BrakeOperation_0 : MC_BR_BrakeOperation;
		MC_ReadActualPosition_0 : MC_ReadActualPosition;
		MC_ReadActualVelocity_0 : MC_ReadActualVelocity;
		MC_SetOverride_0 : MC_SetOverride;
		MC_BR_JogVelocity_0 : MC_BR_JogVelocity;
		MC_BR_InitHome_StpAx_0 : MC_BR_InitHome_StpAx;
		Home_STEP : USINT;
	END_STRUCT;
	ServoLimInternal_typ : 	STRUCT
		STEP : USINT;
		MC_BR_ProcessParID_AcpAx_0 : MC_BR_ProcessParID_AcpAx;
		McAcpAxProcessParIDType_0 : McAcpAxProcessParIDType;
		AktivaciaLimSnimacov_Data : UDINT;
		MC_BR_CyclicProcessParID_AcpAx_0 : MC_BR_CyclicProcessParID_AcpAx;
		McAcpAxCycParIDType_0 : McAcpAxCycParIDType;
		LimSnimace_Data : UDINT;
		KorekcnyCas : TON;
	END_STRUCT;
END_TYPE
```

#### AxisLib.fun - Exported functions and function blocks
```iecst
{REDUND_ERROR} FUNCTION_BLOCK Axis_Servo (*TODO: Add your comment here*) (*$GROUP=User,$CAT=User,$GROUPICON=User.png,$CATICON=User.png*)
	VAR_INPUT
		AxisName : {REDUND_UNREPLICABLE} UDINT;
		CMD : ServoCommand_typ;
		PAR : ServoParametre_typ;
		HomePAR : ServoHomeParametre_typ;
	END_VAR
	VAR_OUTPUT
		STATUS : ServoStatus_typ;
		ErrorDetail : ServoErrorDetail_typ;
	END_VAR
	VAR
		Internal : ServoInternal_typ;
	END_VAR
END_FUNCTION_BLOCK

{REDUND_ERROR} FUNCTION_BLOCK Axis_Krokac (*TODO: Add your comment here*) (*$GROUP=User,$CAT=User,$GROUPICON=User.png,$CATICON=User.png*)
	VAR_INPUT
		AxisName : {REDUND_UNREPLICABLE} UDINT;
		CMD : KrokacCommand_typ;
		PAR : KrokacParametre_typ;
		HomePAR : KrokacHomeParametre_typ;
	END_VAR
	VAR_OUTPUT
		STATUS : KrokacStatus_typ;
		ErrorDetail : KrokacErrorDetail_typ;
	END_VAR
	VAR
		Internal : KrokacInternal_typ;
	END_VAR
END_FUNCTION_BLOCK

{REDUND_ERROR} FUNCTION_BLOCK ServoLim (*TODO: Add your comment here*) (*$GROUP=User,$CAT=User,$GROUPICON=User.png,$CATICON=User.png*)
	VAR_INPUT
		AxisName : UDINT;
		ENABLE : BOOL;
		PositiveLimitSwitch : BOOL;
		NegativeLimitSwitch : BOOL;
		HomingSwitch : BOOL;
	END_VAR
	VAR_OUTPUT
		BUSY : BOOL;
		Error : BOOL;
	END_VAR
	VAR
		Internal : ServoLimInternal_typ;
	END_VAR
END_FUNCTION_BLOCK
```

#### Axis_Servo.st
```iecst
(* TODO: Add your comment here *)
FUNCTION_BLOCK Axis_Servo

	//***********************************************************Power serva*********************************************************************//
	Internal.MC_Power_0.Axis:= AxisName;
	Internal.MC_Power_0.Enable:= CMD.POWER;
	ErrorDetail.Power_Error:= Internal.MC_Power_0.Error;
	ErrorDetail.Power_ErrorID:= Internal.MC_Power_0.ErrorID;
	Internal.MC_Power_0();

	//***********************************************************Zobrazenie stavu serva*********************************************************//
	Internal.MC_ReadAxisInfo_0.Axis:= AxisName;
	Internal.MC_ReadAxisInfo_0.Enable:= TRUE;
	STATUS.ReadyToPower_ON := Internal.MC_ReadAxisInfo_0.ReadyForPowerOn;
	STATUS.Communication_READY:= Internal.MC_ReadAxisInfo_0.CommunicationReady;
	STATUS.Power_ON:= Internal.MC_ReadAxisInfo_0.PowerOn;
	STATUS.Homing_OK:= Internal.MC_ReadAxisInfo_0.IsHomed;
	STATUS.EnableSwitch_ACTIVE:= Internal.MC_ReadAxisInfo_0.AdditionalInfo.DigitalInputStatus.DriveEnable;
	STATUS.HomingSwitch_ACTIVE:= Internal.MC_ReadAxisInfo_0.AdditionalInfo.DigitalInputStatus.HomingSwitch;
	STATUS.NegativeLimitSwitch_ACTIVE:=	Internal.MC_ReadAxisInfo_0.AdditionalInfo.DigitalInputStatus.NegativeLimitSwitch;
	STATUS.PositiveLimitSwitch_ACTIVE:=	Internal.MC_ReadAxisInfo_0.AdditionalInfo.DigitalInputStatus.PositiveLimitSwitch;
	Internal.MC_ReadAxisInfo_0();

	//********************************************************Porucha serva************************************************************************//
	//Zobrazenie poruchy serva//
	Internal.MC_ReadAxisError_0.Axis:= AxisName;
	Internal.MC_ReadAxisError_0.Enable:= CMD.ENABLE;
	STATUS.ERROR_ID:= Internal.MC_ReadAxisError_0.AxisErrorID;
	Internal.MC_ReadAxisError_0();

	Internal.MC_ReadStatus_0.Axis:= AxisName;
	Internal.MC_ReadStatus_0.Enable:= CMD.ENABLE;
	Internal.MC_ReadStatus_0();

	//	IF Internal.MC_Power_0.Error THEN
	//		(*STATUS.ERROR:= TRUE;*)
	IF Internal.MC_Home_0.Error THEN
		STATUS.ERROR:= TRUE;
	ELSIF Internal.MC_BR_JogLimitPosition_0.Error THEN
		STATUS.ERROR:= TRUE;
	ELSIF Internal.MC_BR_JogVelocity_0.Error THEN
		STATUS.ERROR:= TRUE;
	ELSIF Internal.MC_MoveAbsolute_0.Error THEN
		STATUS.ERROR:= TRUE;
	ELSIF Internal.MC_MoveAdditive_0.Error THEN
		STATUS.ERROR:= TRUE;
	ELSIF Internal.MC_MoveVelocity_0.Error THEN
		STATUS.ERROR:= TRUE;
	ELSIF Internal.MC_TorqueControl_0.Error THEN
		STATUS.ERROR:= TRUE;
	ELSIF Internal.MC_Stop_0.Error THEN
		STATUS.ERROR:= TRUE;
	ELSIF Internal.MC_BR_BrakeOperation_0.Error THEN
		STATUS.ERROR:= TRUE;
	ELSIF STATUS.ERROR_ID <> 0 THEN
		STATUS.ERROR:= TRUE;
	ELSE
		STATUS.ERROR:= FALSE;
	END_IF

	//Reset poruchy serva//
	Internal.MC_Reset_0.Axis:= AxisName;
	Internal.MC_Reset_0.Execute:= CMD.ErrorRESET;
	Internal.MC_Reset_0();

	IF CMD.ErrorRESET THEN
		CMD.ENABLE:= FALSE;
	ELSE
		CMD.ENABLE:= TRUE;
	END_IF

	//*********************************************Homing serva***************************************************************************//
	//0 - direct, 1- refrenčný snímač, 2 - limitný snímač, 3 - absolutny encoder, 4 - na moment//
	//Parametre homingu//
	Internal.MC_BR_InitHome_AcpAx_0.Axis:= AxisName;
	Internal.MC_Home_0.Axis:= AxisName;
	IF HomePAR.HomingMode = 0 THEN //Homing na mieste
		Internal.MC_BR_InitHome_AcpAx_0.HomingParameters.HomingMode:= mcHOMING_DIRECT;
	ELSIF HomePAR.HomingMode = 1 THEN //Homing na refernčný snímač
		Internal.MC_BR_InitHome_AcpAx_0.HomingParameters.HomingMode:= mcHOMING_SWITCH_GATE;
		Internal.MC_BR_InitHome_AcpAx_0.HomingParameters.StartDirection:= mcDIR_NEGATIVE;  //Smer hladania refernčného snímača
		Internal.MC_BR_InitHome_AcpAx_0.HomingParameters.SwitchEdge:= mcDIR_NEGATIVE; //Typ hrany referenčného snímača
		Internal.MC_BR_InitHome_AcpAx_0.HomingParameters.HomingDirection:= mcDIR_POSITIVE; //Smer odchodu z referenčného snímača
	ELSIF HomePAR.HomingMode = 2 THEN //Homing na limitný snímač
		Internal.MC_BR_InitHome_AcpAx_0.HomingParameters.HomingMode:= mcHOMING_LIMIT_SWITCH;
		Internal.MC_BR_InitHome_AcpAx_0.HomingParameters.SwitchEdge:= mcDIR_NEGATIVE; //Typ hrany referenčného snímača
		Internal.MC_BR_InitHome_AcpAx_0.HomingParameters.HomingDirection:= mcDIR_POSITIVE; //Smer odchodu z referenčného snímača
	ELSIF  HomePAR.HomingMode = 3 THEN //Homing na absolútny snímač
		Internal.MC_BR_InitHome_AcpAx_0.HomingParameters.HomingMode:= mcHOMING_ABSOLUTE;
	ELSIF HomePAR.HomingMode = 4 THEN //Homing na moment
		Internal.MC_BR_InitHome_AcpAx_0.HomingParameters.HomingMode:= mcHOMING_BLOCK_TORQUE;
		Internal.MC_BR_InitHome_AcpAx_0.HomingParameters.StartDirection:= mcDIR_NEGATIVE;  //Smer hladania refernčného snímača
		Internal.MC_BR_InitHome_AcpAx_0.HomingParameters.SwitchEdge:= mcDIR_NEGATIVE; //Typ hrany referenčného snímača
		Internal.MC_BR_InitHome_AcpAx_0.HomingParameters.HomingDirection:= mcDIR_POSITIVE; //Smer odchodu z referenčného snímača
	ELSE
		Internal.MC_BR_InitHome_AcpAx_0.HomingParameters.HomingMode:= mcHOMING_DIRECT;
	END_IF

	Internal.MC_BR_InitHome_AcpAx_0.HomingParameters.Acceleration:= HomePAR.Acceleration;
	Internal.MC_BR_InitHome_AcpAx_0.HomingParameters.HomingVelocity:= HomePAR.HomingVelocity;
	Internal.MC_BR_InitHome_AcpAx_0.HomingParameters.Position:= HomePAR.Position;
	Internal.MC_BR_InitHome_AcpAx_0.HomingParameters.StartVelocity:= HomePAR.StartVelocity;
	Internal.MC_BR_InitHome_AcpAx_0.HomingParameters.TorqueLimit:= HomePAR.HomeTorque;
	Internal.MC_BR_InitHome_AcpAx_0.HomingParameters.ReferencePulse:= mcSWITCH_OFF;
	Internal.MC_BR_InitHome_AcpAx_0.HomingParameters.KeepDirection:= mcSWITCH_OFF;
	Internal.MC_BR_InitHome_AcpAx_0.HomingParameters.BlockDetectionPositionError:= 1.0;
	Internal.MC_BR_InitHome_AcpAx_0.HomingParameters.PositionErrorStopLimit:= 1.0;
	Internal.MC_Home_0.HomingMode:= mcHOMING_INIT;
	Internal.MC_Home_0.BufferMode:= mcABORTING;
	STATUS.Homing_BUSY:= Internal.MC_Home_0.Busy;
	ErrorDetail.Home_Error:= Internal.MC_Home_0.Error;
	ErrorDetail.Home_ErrorID:= Internal.MC_Home_0.ErrorID;
	Internal.MC_BR_InitHome_AcpAx_0();
	Internal.MC_Home_0();

	CASE Internal.Home_STEP OF

		0: //Nulovanie//
			Internal.MC_BR_InitHome_AcpAx_0.Execute:= FALSE;
			Internal.MC_Home_0.Execute:= FALSE;
			IF NOT CMD.HOME AND NOT Internal.MC_BR_InitHome_AcpAx_0.Error AND NOT Internal.MC_Home_0.Error THEN
				Internal.Home_STEP:= 1;
			END_IF

		1: //Čakanie na spustenie homingu//
			IF CMD.HOME THEN
				Internal.Home_STEP:= 2;
			END_IF

		2: //Načítanie parametrov homingu//
			Internal.MC_BR_InitHome_AcpAx_0.Execute:= TRUE;
			IF Internal.MC_BR_InitHome_AcpAx_0.Error THEN
				Internal.Home_STEP:= 0;
			ELSIF Internal.MC_BR_InitHome_AcpAx_0.Done THEN
				Internal.MC_BR_InitHome_AcpAx_0.Execute:= FALSE;
				Internal.Home_STEP:= 3;
			END_IF

		3: //Spustenie homingu
			Internal.MC_Home_0.Execute:= TRUE;
			IF Internal.MC_Home_0.Error THEN
				Internal.Home_STEP:= 0;
			ELSIF Internal.MC_Home_0.Done THEN
				Internal.Home_STEP:= 0;
			ELSIF NOT CMD.HOME THEN
				Internal.Home_STEP:= 0;
			END_IF
	END_CASE

	//*********************************************Jogging serva**************************************************************************//

	IF (CMD.JoggVPRED OR CMD.JoggVZAD) AND NOT CMD.JoggLimit_ACTIVE AND CMD.ENABLE THEN
		Internal.MC_BR_JogLimitPosition_0.Enable:= FALSE;
		Internal.MC_BR_JogVelocity_0.Enable:= TRUE;
		STATUS.Jogging_BUSY:= Internal.MC_BR_JogVelocity_0.Jogging;
	ELSIF (CMD.JoggVPRED OR CMD.JoggVZAD) AND CMD.JoggLimit_ACTIVE AND CMD.ENABLE THEN
		Internal.MC_BR_JogVelocity_0.Enable:= FALSE;
		Internal.MC_BR_JogLimitPosition_0.Enable:= TRUE;
		STATUS.Jogging_BUSY:= Internal.MC_BR_JogLimitPosition_0.Jogging;
	ELSE
		Internal.MC_BR_JogVelocity_0.Enable:= FALSE;
		Internal.MC_BR_JogLimitPosition_0.Enable:= FALSE;
	END_IF

	//Normálny jogg//
	Internal.MC_BR_JogVelocity_0.Axis:= AxisName;
	Internal.MC_BR_JogVelocity_0.Acceleration:= PAR.JoggAcceleration;
	Internal.MC_BR_JogVelocity_0.Deceleration:= PAR.JoggDeceleration;
	Internal.MC_BR_JogVelocity_0.Velocity:= PAR.JoggVelocity;
	Internal.MC_BR_JogVelocity_0.Jerk:= 0.0;
	Internal.MC_BR_JogVelocity_0.JogPositive:= CMD.JoggVPRED;
	Internal.MC_BR_JogVelocity_0.JogNegative:= CMD.JoggVZAD;
	ErrorDetail.Jogg_Error:= Internal.MC_BR_JogVelocity_0.Error;
	ErrorDetail.Jogg_ErrorID:= Internal.MC_BR_JogVelocity_0.ErrorID;
	Internal.MC_BR_JogVelocity_0();

	//Limitný jogg//
	Internal.MC_BR_JogLimitPosition_0.Axis:= AxisName;
	IF STATUS.ActualPosition >= PAR.JoggPoziciaLimitVPRED THEN
		Internal.MC_BR_JogLimitPosition_0.LastPosition:= STATUS.ActualPosition;
	ELSE
		Internal.MC_BR_JogLimitPosition_0.LastPosition:= PAR.JoggPoziciaLimitVPRED;
	END_IF
	IF STATUS.ActualPosition <= PAR.JoggPoziciaLimitVZAD THEN
		Internal.MC_BR_JogLimitPosition_0.FirstPosition:= STATUS.ActualPosition;
	ELSE
		Internal.MC_BR_JogLimitPosition_0.FirstPosition:= PAR.JoggPoziciaLimitVZAD;
	END_IF
	Internal.MC_BR_JogLimitPosition_0.Acceleration:= PAR.JoggAcceleration;
	Internal.MC_BR_JogLimitPosition_0.Deceleration:= PAR.JoggDeceleration;
	Internal.MC_BR_JogLimitPosition_0.Jerk:= 0.0;
	Internal.MC_BR_JogLimitPosition_0.JogPositive:= CMD.JoggVPRED;
	Internal.MC_BR_JogLimitPosition_0.JogNegative:= CMD.JoggVZAD;
	Internal.MC_BR_JogLimitPosition_0.Velocity:= PAR.JoggVelocity;
	STATUS.JoggLimit_Dosiahnuty:= Internal.MC_BR_JogLimitPosition_0.LimitReached;
	ErrorDetail.JoggLimit_Error:= Internal.MC_BR_JogLimitPosition_0.Error;
	ErrorDetail.JoggLimit_ErrorID:= Internal.MC_BR_JogLimitPosition_0.ErrorID;
	Internal.MC_BR_JogLimitPosition_0();

	//********************************************Move Absolute***************************************************************************//
	Internal.MC_MoveAbsolute_0.Axis:= AxisName;
	Internal.MC_MoveAbsolute_0.Execute:= CMD.MoveAbsolute;
	Internal.MC_MoveAbsolute_0.Acceleration:= PAR.Acceleration;
	Internal.MC_MoveAbsolute_0.Deceleration:= PAR.Deceleration;
	Internal.MC_MoveAbsolute_0.BufferMode:= mcABORTING;
	IF PAR.MoveDirection = 0 THEN
		Internal.MC_MoveAbsolute_0.Direction:= mcDIR_POSITIVE;
	ELSIF PAR.MoveDirection = 1 THEN
		Internal.MC_MoveAbsolute_0.Direction:= mcDIR_NEGATIVE;
	ELSIF PAR.MoveDirection = 10 THEN
		Internal.MC_MoveAbsolute_0.Direction:= mcDIR_BOTH;
	ELSE
		Internal.MC_MoveAbsolute_0.Direction:= 0;
	END_IF
	Internal.MC_MoveAbsolute_0.Jerk:= 0.0;
	Internal.MC_MoveAbsolute_0.Position:= PAR.Position;
	Internal.MC_MoveAbsolute_0.Velocity:= PAR.Velocity;
	STATUS.MoveAbsolute_BUSY:= Internal.MC_MoveAbsolute_0.Busy;
	STATUS.MoveAbsolute_DONE:= Internal.MC_MoveAbsolute_0.Done;
	ErrorDetail.MoveAbsolute_Error:= Internal.MC_MoveAbsolute_0.Error;
	ErrorDetail.MoveAbsolute_ErrorID:= Internal.MC_MoveAbsolute_0.ErrorID;
	Internal.MC_MoveAbsolute_0();

	//********************************************Move Additive*****************************************************************************//
	Internal.MC_MoveAdditive_0.Axis:= AxisName;
	Internal.MC_MoveAdditive_0.Execute:= CMD.MoveAdditive;
	Internal.MC_MoveAdditive_0.Acceleration:= PAR.Acceleration;
	Internal.MC_MoveAdditive_0.Deceleration:= PAR.Deceleration;
	Internal.MC_MoveAdditive_0.Distance:= PAR.AdditivePosition;
	Internal.MC_MoveAdditive_0.Velocity:= PAR.Velocity;
	Internal.MC_MoveAdditive_0.BufferMode:= mcABORTING;
	Internal.MC_MoveAdditive_0.Jerk:= 0.0;
	STATUS.MoveAdditive_BUSY:= Internal.MC_MoveAdditive_0.Busy;
	STATUS.MoveAdditive_DONE:= Internal.MC_MoveAdditive_0.Done;
	ErrorDetail.MoveAdditive_Error:= Internal.MC_MoveAdditive_0.Error;
	ErrorDetail.MoveAdditive_ErrorID:= Internal.MC_MoveAdditive_0.ErrorID;
	Internal.MC_MoveAdditive_0();

	//*********************************************Move Velocity****************************************************************************//
	Internal.MC_MoveVelocity_0.Axis:= AxisName;
	Internal.MC_MoveVelocity_0.Execute:= CMD.MoveVelocity;
	Internal.MC_MoveVelocity_0.Acceleration:= PAR.Acceleration;
	Internal.MC_MoveVelocity_0.Deceleration:= PAR.Deceleration;
	Internal.MC_MoveVelocity_0.BufferMode:= mcABORTING;
	IF PAR.MoveDirection = 0 THEN
		Internal.MC_MoveVelocity_0.Direction:= mcDIR_POSITIVE;
	ELSIF PAR.MoveDirection = 1 THEN
		Internal.MC_MoveVelocity_0.Direction:= mcDIR_NEGATIVE;
	ELSIF PAR.MoveDirection = 10 THEN
		Internal.MC_MoveVelocity_0.Direction:= mcDIR_BOTH;
	ELSE
		Internal.MC_MoveVelocity_0.Direction:= 0;
	END_IF
	Internal.MC_MoveVelocity_0.Velocity:= PAR.Velocity;
	Internal.MC_MoveVelocity_0.Jerk:= 0.0;
	STATUS.MoveVelocity_BUSY:= Internal.MC_MoveVelocity_0.Busy;
	STATUS.Rychlost_Dosiahnuta:= Internal.MC_MoveVelocity_0.InVelocity;
	ErrorDetail.MoveVelocity_Error:= Internal.MC_MoveVelocity_0.Error;
	ErrorDetail.MoveVelocity_ErrorID:= Internal.MC_MoveVelocity_0.ErrorID;
	Internal.MC_MoveVelocity_0();

	//*******************************************Move Torque*******************************************************************************//
	Internal.MC_TorqueControl_0.Axis:= AxisName;
	Internal.MC_TorqueControl_0.Execute:= CMD.MoveTorque;
	Internal.MC_TorqueControl_0.Torque:= PAR.Torque;
	Internal.MC_TorqueControl_0.TorqueRamp:= PAR.TorqueRamp;
	Internal.MC_TorqueControl_0.Velocity:= PAR.TorqueVelocity;
	Internal.MC_TorqueControl_0.Acceleration:= PAR.TorqueAcceleration;
	Internal.MC_TorqueControl_0.Jerk:= 0.0;
	Internal.MC_TorqueControl_0.BufferMode:= mcABORTING;
	STATUS.MoveTorque_BUSY:= Internal.MC_TorqueControl_0.Busy;
	IF PAR.Torque > 0 AND STATUS.MoveTorque_BUSY THEN
		Internal.CasTorque.IN:= (STATUS.ActualTorque >= PAR.Torque);
	ELSIF PAR.Torque < 0 AND STATUS.MoveTorque_BUSY THEN
		Internal.CasTorque.IN:= (STATUS.ActualTorque <= PAR.Torque);
	ELSE
		Internal.CasTorque.IN:= FALSE;
		STATUS.Torque_Dosiahnuty:= FALSE;
	END_IF
	IF Internal.CasTorque.Q THEN
		STATUS.Torque_Dosiahnuty:= TRUE;
	END_IF

	STATUS.Torque_AxisLimit_ACTIVE:= Internal.MC_TorqueControl_0.AxisLimitActive;
	ErrorDetail.MoveTorque_Error:= Internal.MC_TorqueControl_0.Error;
	ErrorDetail.MoveTorque_ErrorID:= Internal.MC_TorqueControl_0.ErrorID;
	Internal.MC_TorqueControl_0();

	Internal.CasTorque.PT:= T#200ms;
	Internal.CasTorque();

	//********************************************Stop serva******************************************************************************//
	Internal.MC_Stop_0.Axis:= AxisName;
	Internal.MC_Stop_0.Execute:= CMD.STOP;
	Internal.MC_Stop_0.Deceleration:= PAR.StopDeceleration;
	Internal.MC_Stop_0.Jerk:= 0.0;
	STATUS.STOP_ACTIVE:= Internal.MC_Stop_0.Done;
	ErrorDetail.Stop_Error:= Internal.MC_Stop_0.Error;
	ErrorDetail.Stop_ErrorID:= Internal.MC_Stop_0.ErrorID;
	Internal.MC_Stop_0();

	//**********************************************Ovládanie brzdy************************************************************************//
	Internal.MC_BR_BrakeOperation_0.Axis:= AxisName;
	IF CMD.UvolniBRZDU THEN
		Internal.MC_BR_BrakeOperation_0.Command:= mcBRAKE_OPEN;
		Internal.MC_BR_BrakeOperation_0.Execute:= TRUE;
		STATUS.UvolnenieBrzdy_DONE:= Internal.MC_BR_BrakeOperation_0.Done;
	ELSIF CMD.ZabrzdiBRZDU THEN
		Internal.MC_BR_BrakeOperation_0.Command:= mcBRAKE_CLOSE;
		Internal.MC_BR_BrakeOperation_0.Execute:= TRUE;
		STATUS.ZabrzdenieBrzdy_DONE:= Internal.MC_BR_BrakeOperation_0.Done;
	ELSE
		Internal.MC_BR_BrakeOperation_0.Execute:= FALSE;
		STATUS.UvolnenieBrzdy_DONE:= FALSE;
		STATUS.ZabrzdenieBrzdy_DONE:= FALSE;
	END_IF
	ErrorDetail.BreakOperation_Error:= Internal.MC_BR_BrakeOperation_0.Error;
	ErrorDetail.BreakOperation_ErrorID:= Internal.MC_BR_BrakeOperation_0.ErrorID;
	Internal.MC_BR_BrakeOperation_0();

	//**********************************************Aktuálna pozícia*************************************************************************//
	Internal.MC_ReadActualPosition_0.Axis:= AxisName;
	Internal.MC_ReadActualPosition_0.Enable:= CMD.ENABLE;
	STATUS.ActualPosition:=	Internal.MC_ReadActualPosition_0.Position;
	Internal.MC_ReadActualPosition_0();

	//**********************************************Aktuálna rýchlosť*************************************************************************//
	Internal.MC_ReadActualVelocity_0.Axis:= AxisName;
	Internal.MC_ReadActualVelocity_0.Enable:= CMD.ENABLE;
	STATUS.ActualVelocity:= Internal.MC_ReadActualVelocity_0.Velocity;
	Internal.MC_ReadActualVelocity_0();

	//**********************************************Aktuálny moment***************************************************************************//
	Internal.MC_ReadActualTorque_0.Axis:= AxisName;
	Internal.MC_ReadActualTorque_0.Enable:= CMD.ENABLE;
	STATUS.ActualTorque:= Internal.MC_ReadActualTorque_0.Torque;
	Internal.MC_ReadActualTorque_0();

	//*********************************************Zmena rýchlosti a rampy********************************************************************//
	Internal.MC_SetOverride_0.Axis:= AxisName;
	Internal.MC_SetOverride_0.Enable:= CMD.UpdatePAR;
	IF PAR.ZmenaRampy < 0.1 THEN
		Internal.MC_SetOverride_0.AccFactor:= 0.1;
	ELSIF PAR.ZmenaRampy > 2.0 THEN
		Internal.MC_SetOverride_0.AccFactor:= 2.0;
	ELSE
		Internal.MC_SetOverride_0.AccFactor:= PAR.ZmenaRampy;
	END_IF
	IF PAR.ZmenaRychlosti < 0.1 THEN
		Internal.MC_SetOverride_0.VelFactor:= 0.1;
	ELSIF PAR.ZmenaRychlosti > 2.0 THEN
		Internal.MC_SetOverride_0.VelFactor:= 2.0;
	ELSE
		Internal.MC_SetOverride_0.VelFactor:= PAR.ZmenaRychlosti;
	END_IF
	STATUS.UpdatePAR_DONE:= Internal.MC_SetOverride_0.Enabled;
	Internal.MC_SetOverride_0();

END_FUNCTION_BLOCK
```
